(* PLC project Horosheva_14_20160824, CODESYS CODESYS V3.5 SP21 *)
(* stored: creationDateTime 2025-03-30T00:33:44.49212, version 0.0.0.107, modificationDateTime 2025-03-30T00:32:10.5601067 *)

TYPE VLV : STRUCT
  CW : VLV_CW;
  SW : VLV_SW;
  rSetPos : REAL;
  rActPos : REAL;
  wStatus : WORD;
  res7 : INT;
  res8 : INT;
  res9 : INT;
  res10 : INT;
  res11 : INT;
  res12 : INT;
  res13 : INT;
  res14 : INT;
  res15 : INT;
END_STRUCT;
END_TYPE

TYPE MTR : STRUCT
  CW : MTR_CW;
  SW : MTR_SW;
  rMinFreq : REAL;
  rMaxFreq : REAL;
  rManFreq : REAL;
  rAutoFreq : REAL;
  rActFreq : REAL;
  rCurrent : REAL;
  rRunHours : REAL;
  rkWhCount : REAL;
  enStatus : MTR_Stat;
  wFC_StatusWord : WORD;
  dwFC_AlarmWord : DWORD;
  dwFC_WarnWord : DWORD;
  wFC_ErrCode : WORD;
  wIndex : WORD;
  rPower : REAL;
  rHeatsinkTemp : REAL;
  res3 : REAL;
END_STRUCT;
END_TYPE

TYPE SNSR_SW : STRUCT
  Fault : BIT;
  HH_alarm : BIT;
  HL_alarm : BIT;
  LH_alarm : BIT;
  LL_alarm : BIT;
  res5 : BIT;
  res6 : BIT;
  res7 : BIT;
  res8 : BIT;
  res9 : BIT;
  res10 : BIT;
  res11 : BIT;
  res12 : BIT;
  res13 : BIT;
  res14 : BIT;
  res15 : BIT;
END_STRUCT;
END_TYPE

TYPE SNSR_CW : STRUCT
  LimEn : BIT;
  FltrEn : BIT;
  SimEn : BIT;
  ExtFault : BIT;
  res4 : BIT;
  res5 : BIT;
  res6 : BIT;
  res7 : BIT;
  bar_kgf : BIT;
  res9 : BIT;
  res10 : BIT;
  res11 : BIT;
  res12 : BIT;
  res13 : BIT;
  res14 : BIT;
  res15 : BIT;
END_STRUCT;
END_TYPE

TYPE SNSR : STRUCT
  CW : SNSR_CW;
  SW : SNSR_SW;
  k : REAL;
  b : REAL;
  ADC_Range : INT;
  SamplingTime : INT;
  HH : REAL;
  HL : REAL;
  LH : REAL;
  LL : REAL;
  DeadBand : REAL;
  LimDelay : INT;
  res19 : INT;
  res20 : INT;
  res21 : INT;
  PIW : INT;
  IntValue : INT;
  RealValue : REAL;
  SimValue : REAL;
  AccumDir : REAL;
  AccumRev : REAL;
END_STRUCT;
END_TYPE

TYPE VLV_SW : STRUCT
  xRem : BIT;
  xManAuto : BIT;
  xCOM_Open : BIT;
  xCOM_Close : BIT;
  xRUN : BIT;
  xOpened : BIT;
  xClosed : BIT;
  xAlarmAccum : BIT;
  xManOK : BIT;
  xAutoOK : BIT;
  xRunManual : BIT;
  xRunAuto : BIT;
  res12 : BIT;
  res13 : BIT;
  res14 : BIT;
  res15 : BIT;
END_STRUCT;
END_TYPE

(* values of VLV_Stat: STANDBY: Standby; OPENED: Opened; CLOSED: Closed; ALARM_ACCUM: Alarm; BLOCK: Blocked (QM off or smth. else) *)

TYPE VLV_Stat : (STANDBY := 0, OPENED := 1, CLOSED := 2, ALARM_ACCUM := 3, BLOCK := 4);
END_TYPE

TYPE VLV_CW : STRUCT
  xEnable : BIT;
  xAuxON : BIT;
  xExtraAlarm : BIT;
  xACK : BIT;
  xAutoMode : BIT;
  xManMode : BIT;
  xManOpen : BIT;
  xStop : BIT;
  xManClose : BIT;
  xAutoOpen : BIT;
  xAutoClose : BIT;
  xExtraEn : BIT;
  res12 : BIT;
  res13 : BIT;
  res14 : BIT;
  xSimEn : BIT;
END_STRUCT;
END_TYPE

(* values of MTR_Stat: STANDBY: Standby; RUN_MAN: Work in manual mode; STAND_MAN: Stand in manual mode; RUN_AUTO: Work in auto mode; STAND_AUTO: Stand in auto mode; NOT_IN_CYCLE: In auto mode, but not in auto cycle; ALARM_ACCUM: Alarm; BLOCK: Blocked (QM off or smth. else) *)

(* -----Motor status-----// *)
TYPE MTR_Stat : (STANDBY := 0, RUN_MAN := 1, STAND_MAN := 2, RUN_AUTO := 3, STAND_AUTO := 5, NOT_IN_CYCLE := 4, ALARM_ACCUM := 6, BLOCK := 7);
END_TYPE

TYPE MTR_CW : STRUCT
  xEnable : BIT;
  xAuxON : BIT;
  xExtraAlarm : BIT;
  xACK : BIT;
  xAutoMode : BIT;
  xManMode : BIT;
  xManStart : BIT;
  xManStop : BIT;
  xAutoON : BIT;
  xExtraEn : BIT;
  res10 : BIT;
  res11 : BIT;
  res12 : BIT;
  res13 : BIT;
  res14 : BIT;
  xSimEn : BIT;
END_STRUCT;
END_TYPE

TYPE MTR_SW : STRUCT
  xRem : BIT;
  xManAuto : BIT;
  xRUN : BIT;
  xCOM : BIT;
  xAlarmAccum : BIT;
  xReady : BIT;
  res6 : BIT;
  res7 : BIT;
  xManOK : BIT;
  xAutoOK : BIT;
  xRunManual : BIT;
  xRunAuto : BIT;
  res12 : BIT;
  res13 : BIT;
  res14 : BIT;
  res15 : BIT;
END_STRUCT;
END_TYPE

TYPE CCL_WRN : STRUCT
  xVoltageOK : BIT;
  xPLC_ConectOK : BIT;
  xSecurity : BIT;
  xFire : BIT;
  xFireEqipFault : BIT;
  xDrainLL : BIT;
  xDrainHL : BIT;
  xDrainHH : BIT;
  xPMP1_Dry : BIT;
  xPMP2_Dry : BIT;
  xPMP3_Dry : BIT;
  res11 : BIT;
  res12 : BIT;
  res13 : BIT;
  res14 : BIT;
  res15 : BIT;
  res16 : BIT;
  res17 : BIT;
  res18 : BIT;
  res19 : BIT;
  res20 : BIT;
  res21 : BIT;
  res22 : BIT;
  res23 : BIT;
  res24 : BIT;
  res25 : BIT;
  res26 : BIT;
  res27 : BIT;
  res28 : BIT;
  res29 : BIT;
  res30 : BIT;
  res31 : BIT;
END_STRUCT;
END_TYPE

TYPE CCL : STRUCT
  CW : CCL_CW;
  SW : CCL_SW;
  WRN : CCL_WRN;
  uiRotHour : UINT;
  uiRotMin : UINT;
  res6 : WORD;
  res7 : WORD;
  rSP : REAL;
  PmpConnFreq : REAL;
  PmpDisconnFreq : REAL;
  res11 : REAL;
END_STRUCT;
END_TYPE

TYPE CCL_SW : STRUCT
  xALARM : BIT;
  xON : BIT;
  xRunning : BIT;
  res3 : BIT;
  res4 : BIT;
  res5 : BIT;
  res6 : BIT;
  res7 : BIT;
  res8 : BIT;
  res9 : BIT;
  res10 : BIT;
  res11 : BIT;
  res12 : BIT;
  res13 : BIT;
  res14 : BIT;
  res15 : BIT;
END_STRUCT;
END_TYPE

TYPE CCL_CW : STRUCT
  xAuxON : BIT;
  xStart : BIT;
  xStop : BIT;
  xPulseStart : BIT;
  xACK : BIT;
  res5 : BIT;
  res6 : BIT;
  res7 : BIT;
  xAuxStop : BIT;
  xPmpRot : BIT;
  res10 : BIT;
  res11 : BIT;
  res12 : BIT;
  res13 : BIT;
  res14 : BIT;
  res15 : BIT;
END_STRUCT;
END_TYPE

TYPE PID_SW : STRUCT
  Error : BIT;
  LL : BIT;
  LH : BIT;
  res3 : BIT;
  res4 : BIT;
  res5 : BIT;
  res6 : BIT;
  res7 : BIT;
  res8 : BIT;
  res9 : BIT;
  res10 : BIT;
  res11 : BIT;
  res12 : BIT;
  res13 : BIT;
  res14 : BIT;
  res15 : BIT;
END_STRUCT;
END_TYPE

TYPE PID_CW : STRUCT
  En : BIT;
  ManMode : BIT;
  Reset : BIT;
  Hold : BIT;
  res4 : BIT;
  res5 : BIT;
  res6 : BIT;
  res7 : BIT;
  res8 : BIT;
  res9 : BIT;
  res10 : BIT;
  res11 : BIT;
  res12 : BIT;
  res13 : BIT;
  res14 : BIT;
  res15 : BIT;
END_STRUCT;
END_TYPE

TYPE PID_ : STRUCT
  CW : PID_CW;
  SW : PID_SW;
  SetPoint : REAL;
  Kp : REAL;
  Tn : REAL;
  Tv : REAL;
  Td : REAL;
  Offset : REAL;
  ManVal : REAL;
  LL : REAL;
  LH : REAL;
  Y : REAL;
  DIFF : REAL;
  ActValue : REAL;
  DeadBand : REAL;
  MinStop : TIME;
  MinWork : TIME;
END_STRUCT;
END_TYPE

TYPE SP_SW : STRUCT
  xManual : BIT;
  xSched : BIT;
  xRemote : BIT;
  res3 : BIT;
  res4 : BIT;
  res5 : BIT;
  res6 : BIT;
  res7 : BIT;
  res8 : BIT;
  res9 : BIT;
  res10 : BIT;
  res11 : BIT;
  res12 : BIT;
  res13 : BIT;
  res14 : BIT;
  res15 : BIT;
END_STRUCT;
END_TYPE

TYPE SP : STRUCT
  CW : SP_CW;
  SW : SP_SW;
  wSPLocSetNum : WORD;
  wSPLocCurrNum : WORD;
  sSPDate : SP_Date;
  sSPLocSet : SP_Loc;
  arrSPLocCurr : ARRAY[1..4] OF SP_Loc;
  rSPRem : REAL;
  wConnect : WORD;
  wSPRemSet : WORD;
END_STRUCT;
END_TYPE

TYPE SP_Loc : STRUCT
  wHour : WORD;
  wMinute : WORD;
  rSP : REAL;
END_STRUCT;
END_TYPE

TYPE SP_Date : STRUCT
  wSummMonth : WORD;
  wSummDay : WORD;
  wWinMonth : WORD;
  wWinDay : WORD;
END_STRUCT;
END_TYPE

TYPE SP_CW : STRUCT
  xManMode : BIT;
  xAutoLocMode : BIT;
  xAutoRemMode : BIT;
  xConnect : BIT;
  xSPLocSet : BIT;
  xSPRemSet : BIT;
  res6 : BIT;
  res7 : BIT;
  res8 : BIT;
  res9 : BIT;
  res10 : BIT;
  res11 : BIT;
  res12 : BIT;
  res13 : BIT;
  res14 : BIT;
  res15 : BIT;
END_STRUCT;
END_TYPE

VAR_GLOBAL  (* GVL *)
  i_write_set_point_Pump : BOOL;
  ETH_Set_ip : SEC_ETH_UTIL.changeIPAddress;
  wSecond AT %MW41605 : UINT;
  wYear AT %MW41600 : UINT;
  wMonth AT %MW41601 : UINT;
  wDay AT %MW41602 : UINT;
  wHour AT %MW41603 : UINT;
  wMinute AT %MW41604 : UINT;
  x_Set_ip : BOOL;
  x_Save_ip : BOOL;
  xPLC_RUN : BOOL;
  i_ADC_Range : INT := 10000;
  PLC_Cycle : REAL := 0.1;
  i_Set_Point_Pressure AT %MD576 : REAL;
  i_input_ip_address AT %MB500 : ARRAY[1..4] OF BYTE;
  FirstCycle : BOOL;
END_VAR

PROGRAM CycleSect
  VAR
    PLC_RUN : BOOL;
    CycleDelay : TON;
    PulseStart : R_TRIG;
    xVoltageOK : BOOL;
    xExtAlarm : BOOL;
    PLS_RESET : R_TRIG;
  END_VAR

            
PLC_RUN:= (PLC_R.i_wStatus = 16#0002);
PLS_RESET(CLK:= PLC_RUN);

Cycle.CW.xAuxON:= PLC_RUN;
Cycle.SW.xON:= (Cycle.CW.xStart OR Cycle.SW.xON) AND NOT Cycle.CW.xAuxStop;  

CycleDelay(IN:= Cycle.SW.xON,PT:= T#3S);
PulseStart(CLK:= CycleDelay.Q AND (Cycle.CW.xStart OR NOT Cycle.SW.xRunning), Q=> Cycle.CW.xPulseStart);

Cycle.SW.xRunning:= CycleDelay.Q;
				
Cycle.CW.xStart:= FALSE;
IF Cycle.CW.xAuxStop THEN
	Cycle.CW.xStop:= FALSE;
	Cycle.CW.xAuxStop:= FALSE;
END_IF



          
END_PROGRAM

PROGRAM CtrlSect
  VAR
    xPMP2_StartRdy : BOOL;
    xPMP3_StartRdy : BOOL;
    xPMP1_StartRdy : BOOL;
    xPMP1_StopRdy : BOOL;
    xPMP2_StopRdy : BOOL;
    xPMP3_StopRdy : BOOL;
    StartPulse : R_TRIG;
    AuxPmpOnTmr : TON;
    AuxPmpOnPls : R_TRIG;
    xStartAuxPmpReq : BOOL;
    AuxPmpOffTmr : TON;
    AuxPmpOffPls : R_TRIG;
    xStopAuxPmpReq : BOOL;
    MainReg : PID;
    AuxReg : PID;
    MainPID_SetFreq : REAL;
    AuxPID_SetFreq : REAL;
    PMP1_Rising : BOOL;
    PMP2_Rising : BOOL;
    PMP3_Rising : BOOL;
    CyclicSubTimer : TON;
    CyclicSubPls : R_TRIG;
    AuxPmpOnTmrET : TIME;
    AuxPmpOffTmrET : TIME;
    iRunPmpNum : INT;
    MainReg_Ymin : REAL;
    AuxReg_Ymin : REAL;
    RotReq : BOOL;
    ConnPls : R_TRIG;
    DisconnPls : R_TRIG;
  END_VAR

            //=====================================================================================================================//
// Definition of pumps ready to start
//=====================================================================================================================//
xPMP1_StartRdy:= PMP1.SW.xAutoOK AND NOT PMP1.SW.xRUN AND
				((PMP1_WorkTimer[3] <= PMP2_WorkTimer[3]) OR NOT PMP2.SW.xAutoOK OR PMP2.SW.xRUN) AND
				((PMP1_WorkTimer[3] <= PMP3_WorkTimer[3]) OR NOT PMP3.SW.xAutoOK OR PMP3.SW.xRUN);
xPMP2_StartRdy:= PMP2.SW.xAutoOK AND NOT PMP2.SW.xRUN AND
				((PMP2_WorkTimer[3] <= PMP1_WorkTimer[3]) OR NOT PMP1.SW.xAutoOK OR PMP1.SW.xRUN) AND 
				((PMP2_WorkTimer[3] <= PMP3_WorkTimer[3]) OR NOT PMP3.SW.xAutoOK OR PMP3.SW.xRUN);
xPMP3_StartRdy:= PMP3.SW.xAutoOK AND NOT PMP3.SW.xRUN AND 
				((PMP3_WorkTimer[3] <= PMP1_WorkTimer[3]) OR NOT PMP1.SW.xAutoOK OR PMP1.SW.xRUN) AND 
				((PMP3_WorkTimer[3] <= PMP2_WorkTimer[3]) OR NOT PMP2.SW.xAutoOK OR PMP2.SW.xRUN);

//=====================================================================================================================//
// Identifying a pump ready to stop
//=====================================================================================================================//
xPMP1_StopRdy:= PMP1.SW.xAutoOK AND PMP1.SW.xRUN AND 
				((PMP1_WorkTimer[3] >= PMP2_WorkTimer[3]) OR NOT PMP2.SW.xRUN) AND 
				((PMP1_WorkTimer[3] >= PMP3_WorkTimer[3]) OR NOT PMP3.SW.xRUN);
xPMP2_StopRdy:= PMP2.SW.xAutoOK AND PMP2.SW.xRUN AND 
				((PMP2_WorkTimer[3] >= PMP1_WorkTimer[3]) OR NOT PMP1.SW.xRUN) AND 
				((PMP2_WorkTimer[3] >= PMP3_WorkTimer[3]) OR NOT PMP3.SW.xRUN);
xPMP3_StopRdy:= PMP3.SW.xAutoOK AND PMP3.SW.xRUN AND 
				((PMP3_WorkTimer[3] >= PMP1_WorkTimer[3]) OR NOT PMP1.SW.xRUN) AND 
				((PMP3_WorkTimer[3] >= PMP2_WorkTimer[3]) OR NOT PMP2.SW.xRUN);
				
//=====================================================================================================================//
// Determining the number of operating pumps and the minimum output value of the main PID controller
//=====================================================================================================================//
IF (PMP1.SW.xRUN AND PMP1.SW.xAutoOK) AND (PMP2.SW.xRUN AND PMP2.SW.xAutoOK) AND(PMP3.SW.xRUN AND PMP3.SW.xAutoOK) THEN
	MainReg_Ymin:= MAX(MAX(PMP1.rMinFreq, PMP2.rMinFreq), PMP3.rMinFreq);
	iRunPmpNum:= 3;
ELSIF ((PMP1.SW.xRUN AND PMP1.SW.xAutoOK) AND (PMP2.SW.xRUN AND PMP2.SW.xAutoOK)) THEN
	MainReg_Ymin:= MAX(PMP1.rMinFreq, PMP2.rMinFreq);
	iRunPmpNum:= 2;
ELSIF ((PMP1.SW.xRUN AND PMP1.SW.xAutoOK) AND (PMP3.SW.xRUN AND PMP3.SW.xAutoOK)) THEN
	MainReg_Ymin:= MAX(PMP1.rMinFreq, PMP3.rMinFreq);
	iRunPmpNum:= 2; 
ELSIF ((PMP2.SW.xRUN AND PMP2.SW.xAutoOK) AND (PMP3.SW.xRUN AND PMP3.SW.xAutoOK)) THEN
	MainReg_Ymin:= MAX(PMP2.rMinFreq, PMP3.rMinFreq);
	iRunPmpNum:= 2;
ELSIF (PMP1.SW.xRUN AND PMP1.SW.xAutoOK) THEN
	MainReg_Ymin:= PMP1.rMinFreq;
	iRunPmpNum:= 1;
ELSIF (PMP2.SW.xRUN AND PMP2.SW.xAutoOK) THEN
	MainReg_Ymin:= PMP2.rMinFreq;
	iRunPmpNum:= 1;
ELSIF (PMP3.SW.xRUN AND PMP3.SW.xAutoOK) THEN
	MainReg_Ymin:= PMP3.rMinFreq;
	iRunPmpNum:= 1;
ELSE
	MainReg_Ymin:= 25.0;
	iRunPmpNum:= 0;
END_IF
			
//====================================================================================================================//
// Pump start request condition
//====================================================================================================================//
AuxPmpOnTmr(IN:= ((PMP1.rActFreq >= (PMP1.rMaxFreq - 1.0)) OR
				  (PMP2.rActFreq >= (PMP2.rMaxFreq - 1.0)) OR
				  (PMP3.rActFreq >= (PMP3.rMaxFreq - 1.0))) AND (xPMP1_StartRdy OR xPMP2_StartRdy OR xPMP3_StartRdy) AND
				 ((BP01.RealValue + 0.3) <= Cycle.rSP) AND Cycle.SW.xRunning, PT:= T#180S, ET=> AuxPmpOnTmrET);
AuxPmpOnPls(CLK:= AuxPmpOnTmr.Q);
//====================================================================================================================//
// Pump shutdown request condition
//====================================================================================================================//
AuxPmpOffTmr(IN:= (((PMP1.rActFreq < Cycle.PmpDisconnFreq) AND xPMP1_StopRdy) OR
				  ((PMP2.rActFreq < Cycle.PmpDisconnFreq) AND xPMP2_StopRdy) OR
				  ((PMP3.rActFreq < Cycle.PmpDisconnFreq) AND xPMP3_StopRdy)) AND (iRunPmpNum > 1) AND
				  ((BP01.RealValue + 0.2) >= Cycle.rSP) AND Cycle.SW.xRunning, PT:= T#180S, ET=> AuxPmpOffTmrET);
AuxPmpOffPls(CLK:= AuxPmpOffTmr.Q);
//====================================================================================================================//
// Time rotation of pumps
//====================================================================================================================//
IF Cycle.CW.xPmpRot AND (xPMP1_StartRdy OR xPMP2_StartRdy OR xPMP3_StartRdy) AND (PLC_RTC.wHour = Cycle.uiRotHour) AND (PLC_RTC.wMinute = Cycle.uiRotMin) AND (PLC_RTC.wSecond = 1) THEN
	RotReq:= TRUE;
END_IF

IF DisconnPls.Q OR NOT Cycle.CW.xPmpRot OR ((PMP1_Rising AND PMP1.SW.xAlarmAccum) OR (PMP2_Rising AND PMP2.SW.xAlarmAccum) OR (PMP3_Rising AND PMP3.SW.xAlarmAccum) AND NOT (xPMP1_StartRdy OR xPMP2_StartRdy OR xPMP3_StartRdy)) THEN
	RotReq:= FALSE;
END_IF

ConnPls(CLK:= RotReq);
DisconnPls(CLK:= RotReq AND (AuxPID.Y >= MainPID.Y));
//====================================================================================================================//
// Generation of pump start-up and shutdown requests
//====================================================================================================================//
StartPulse(CLK:= Cycle.SW.xRunning);
IF Cycle.SW.xRunning THEN
	IF StartPulse.Q OR AuxPmpOnPls.Q OR (iRunPmpNum = 0) OR ConnPls.Q OR (PMP1_Rising AND PMP1.SW.xAlarmAccum) OR (PMP2_Rising AND PMP2.SW.xAlarmAccum) OR (PMP3_Rising AND PMP3.SW.xAlarmAccum) THEN
		xStartAuxPmpReq:= TRUE;
	END_IF

	IF (AuxPmpOffPls.Q OR DisconnPls.Q) AND (iRunPmpNum > 1) THEN
		xStopAuxPmpReq:= TRUE;
	END_IF

ELSE	
	xStartAuxPmpReq:= FALSE;
	xStopAuxPmpReq:= FALSE;
	PMP1.CW.xAutoON:= FALSE;
	PMP2.CW.xAutoON:= FALSE;
	PMP3.CW.xAutoON:= FALSE;
	PMP1_Rising:= FALSE;
	PMP2_Rising:= FALSE;
	PMP3_Rising:= FALSE;
	RotReq:= FALSE;
END_IF

//====================================================================================================================//
// Formation of an acceleration bit on request to start a pump unit or connect an additional pump
//====================================================================================================================//
IF xStartAuxPmpReq THEN
	IF xPMP1_StartRdy THEN
		PMP1_Rising:= TRUE;
	ELSIF xPMP2_StartRdy THEN
		PMP2_Rising:= TRUE;
	ELSIF xPMP3_StartRdy THEN
		PMP3_Rising:= TRUE;
	END_IF
	xStartAuxPmpReq:= FALSE;
END_IF
//====================================================================================================================//
// Setpoint reduction on acceleration
//====================================================================================================================//
IF PMP1_Rising OR PMP2_Rising OR PMP3_Rising THEN
	MainPID.SetPoint:= Cycle.rSP - 1.0;			
	AuxPID.SetPoint:= Cycle.rSP;				
ELSE
	MainPID.SetPoint:= Cycle.rSP;
	AuxPID.SetPoint:= 0.0;
END_IF
//====================================================================================================================//
// Pump No. 1 run-up
//====================================================================================================================// 	
IF PMP1_Rising THEN														
	PMP1.CW.xAutoON:= TRUE;													
	PMP1.rAutoFreq:= AuxPID_SetFreq;										
	                                                                              
	IF AuxPID.Y >= MainPID.Y OR PMP1.SW.xAlarmAccum THEN					
		PMP1_Rising:= FALSE;												
	END_IF                                                                        
ELSIF NOT (xStopAuxPmpReq AND xPMP1_StopRdy) AND NOT Cycle.CW.xStop THEN	 
	PMP1.rAutoFreq:= MainPID_SetFreq;										
END_IF
//====================================================================================================================//
// Pump No. 2 run-up
//====================================================================================================================//
IF PMP2_Rising THEN
	PMP2.CW.xAutoON:= TRUE;
	PMP2.rAutoFreq:= AuxPID_SetFreq;		
	
	IF AuxPID.Y >= MainPID.Y OR PMP2.SW.xAlarmAccum THEN
		PMP2_Rising:= FALSE;
	END_IF
ELSIF NOT (xStopAuxPmpReq AND xPMP2_StopRdy) AND NOT Cycle.CW.xStop THEN
	PMP2.rAutoFreq:= MainPID_SetFreq;
END_IF
//====================================================================================================================//
// Pump No. 3 run-up
//====================================================================================================================//
IF PMP3_Rising THEN
	PMP3.CW.xAutoON:= TRUE;
	PMP3.rAutoFreq:= AuxPID_SetFreq;		

	IF AuxPID.Y >= MainPID.Y OR PMP3.SW.xAlarmAccum THEN
		PMP3_Rising:= FALSE;
	END_IF
ELSIF NOT (xStopAuxPmpReq AND xPMP3_StopRdy) AND NOT Cycle.CW.xStop THEN
	PMP3.rAutoFreq:= MainPID_SetFreq;
END_IF

//====================================================================================================================//
// Smooth stop of redundant pump
//====================================================================================================================//
CyclicSubTimer(IN:= NOT CyclicSubTimer.Q, PT:= T#5S);
CyclicSubPls(CLK:= CyclicSubTimer.Q);

IF xStopAuxPmpReq  THEN
	IF xPMP1_StopRdy THEN
		IF CyclicSubPls.Q THEN
			PMP1.rAutoFreq:= PMP1.rAutoFreq - 2.0;
		END_IF
		IF PMP1.rActFreq <= PMP1.rMinFreq + 2.0 THEN
			PMP1.CW.xAutoON:= FALSE;
			xStopAuxPmpReq:= FALSE;
		END_IF
	ELSIF xPMP2_StopRdy THEN
		IF CyclicSubPls.Q THEN
			PMP2.rAutoFreq:= PMP2.rAutoFreq - 2.0;
		END_IF
		IF PMP2.rActFreq <= PMP2.rMinFreq + 2.0 THEN
			PMP2.CW.xAutoON:= FALSE;
			xStopAuxPmpReq:= FALSE;
		END_IF
	ELSIF xPMP3_StopRdy THEN
		IF CyclicSubPls.Q THEN
			PMP3.rAutoFreq:= PMP3.rAutoFreq - 2.0;
		END_IF
		IF PMP3.rActFreq <= PMP3.rMinFreq + 2.0 THEN
			PMP3.CW.xAutoON:= FALSE;
			xStopAuxPmpReq:= FALSE;
		END_IF
	END_IF
END_IF

//====================================================================================================================//
// Resetting the start command in automatic cycle if the pump is not in automatic mode
//====================================================================================================================//
IF NOT PMP1.SW.xAutoOK THEN
	PMP1.CW.xAutoON:= FALSE;
END_IF	
IF NOT PMP2.SW.xAutoOK THEN
	PMP2.CW.xAutoON:= FALSE;
END_IF	
IF NOT PMP3.SW.xAutoOK THEN
	PMP3.CW.xAutoON:= FALSE;
END_IF	

//====================================================================================================================//
// Soft stop of pumps to disable automatic cycle
//====================================================================================================================//
IF Cycle.CW.xStop AND Cycle.SW.xRunning THEN
	xStartAuxPmpReq:= FALSE;
	xStopAuxPmpReq:= FALSE;
	IF CyclicSubPls.Q THEN
		PMP1.rAutoFreq:= PMP1.rAutoFreq - 2.0;
		PMP2.rAutoFreq:= PMP2.rAutoFreq - 2.0;
		PMP3.rAutoFreq:= PMP3.rAutoFreq - 2.0;
	END_IF
	
	IF ((PMP1.rActFreq <= PMP1.rMinFreq + 2.0) OR NOT PMP1.SW.xAutoOK) AND 
		((PMP2.rActFreq <= PMP2.rMinFreq + 2.0) OR NOT PMP2.SW.xAutoOK) AND 
		((PMP3.rActFreq <= PMP3.rMinFreq + 2.0) OR NOT PMP3.SW.xAutoOK) THEN
		Cycle.CW.xAuxStop:= TRUE;
	END_IF
END_IF

//====================================================================================================================//
// Determining the minimum output value of the auxiliary PID controller
//====================================================================================================================//
IF PMP1_Rising THEN
	AuxReg_Ymin:= PMP1.rMinFreq;
ELSIF PMP2_Rising THEN
	AuxReg_Ymin:= PMP2.rMinFreq;
ELSIF PMP3_Rising THEN
	AuxReg_Ymin:= PMP3.rMinFreq;
ELSE
	AuxReg_Ymin:= 25.0;
END_IF

//====================================================================================================================//
// Main PID controller
//====================================================================================================================//
MainPID.CW.Reset:= NOT(Cycle.SW.xRunning AND (PMP1.SW.xRunAuto OR PMP2.SW.xRunAuto OR PMP3.SW.xRunAuto));
MainPID.ActValue:= BP01.RealValue;
MainReg(
	ACTUAL:= MainPID.ActValue, 
	SET_POINT:= MainPID.SetPoint, 
	KP:= MainPID.Kp, 
	TN:= MainPID.Tn, 
	TV:= MainPID.Tv, 
	Y_MANUAL:= MainPID.ManVal, 
	Y_OFFSET:= MainPID.Offset, 
	Y_MIN:= MainReg_Ymin * 10.0,
	Y_MAX:= 500.0, 
	MANUAL:= MainPID.CW.ManMode, 
	RESET:= MainPID.CW.Reset, 
	Y=> MainPID.Y, 
	LIMITS_ACTIVE=> , 
	OVERFLOW=> );
MainPID_SetFreq:= MainPID.Y / 10.0; 

//====================================================================================================================//
// Auxiliary PID controller used to accelerate the auxiliary pump
//====================================================================================================================//	
AuxPID.CW.Reset:= NOT(Cycle.SW.xRunning AND (PMP1_Rising OR PMP2_Rising OR PMP3_Rising));	
AuxPID.ActValue:= BP01.RealValue;
AuxReg(
	ACTUAL:= AuxPID.ActValue, 
	SET_POINT:= AuxPID.SetPoint, 
	KP:= AuxPID.Kp, 
	TN:= AuxPID.Tn, 
	TV:= AuxPID.Tv, 
	Y_MANUAL:= AuxPID.ManVal, 
	Y_OFFSET:= AuxPID.Offset, 
	Y_MIN:= AuxReg_Ymin * 10.0,
	Y_MAX:= 500.0, 
	MANUAL:= AuxPID.CW.ManMode, 
	RESET:= AuxPID.CW.Reset, 
	Y=> AuxPID.Y, 
	LIMITS_ACTIVE=> , 
	OVERFLOW=> );
AuxPID_SetFreq:= AuxPID.Y / 10.0;
	
	
	
	
	
	
	
	
          
END_PROGRAM

FUNCTION_BLOCK MotorFB
  VAR_INPUT
    SetOvertime : TIME;
    Cycle : CCL;
  END_VAR
  VAR_OUTPUT
    rFreqValue : REAL;
    WorkTime : ARRAY[1..4] OF UDINT;
  END_VAR
  VAR_IN_OUT
    Mot_strct : MTR;
  END_VAR
  VAR
    TON_Overtime : TON;
    xAlarmFeedback : BOOL;
    xEnableMotorAuto : BOOL;
    xCOM : BOOL;
    WTC : WTCount;
    xAlarmBlock : BOOL;
  END_VAR

            	(*Alarm Feedback processing*)
TON_Overtime(IN:=Mot_strct.CW.xEnable AND ((Mot_strct.SW.xCOM AND NOT Mot_strct.SW.xRUN) OR (NOT Mot_strct.SW.xCOM AND Mot_strct.SW.xRUN)),PT:=SetOvertime);

IF TON_Overtime.Q THEN
	xAlarmFeedback:=TRUE;
END_IF; 

IF NOT Mot_strct.CW.xExtraEn AND xCOM THEN
	xAlarmBlock:= TRUE;
END_IF

Mot_strct.SW.xAlarmAccum:= xAlarmFeedback OR Mot_strct.CW.xExtraAlarm OR xAlarmBlock;

IF Mot_strct.CW.xACK THEN
	xAlarmFeedback:= FALSE;
	xAlarmBlock:= FALSE;
END_IF
	
	(*Auto/Manual mode selection*)
IF Mot_strct.CW.xAutoMode THEN
	xEnableMotorAuto:= TRUE;
ELSIF Mot_strct.CW.xManMode THEN
	xEnableMotorAuto:= FALSE;
END_IF;
Mot_strct.SW.xManAuto:= xEnableMotorAuto; 

Mot_strct.SW.xManOK:= NOT Mot_strct.SW.xAlarmAccum AND Mot_strct.CW.xAuxON AND Mot_strct.CW.xEnable AND NOT xEnableMotorAuto;
Mot_strct.SW.xAutoOK:= NOT Mot_strct.SW.xAlarmAccum AND Mot_strct.CW.xAuxON AND Mot_strct.CW.xEnable AND xEnableMotorAuto;

	(*Motor ready to start*)
Mot_strct.SW.xReady:= (Mot_strct.SW.xManOK OR Mot_strct.SW.xAutoOK) AND NOT Mot_strct.SW.xAlarmAccum;

	(*Manual mode activation*)
IF Mot_strct.CW.xManStart THEN
	Mot_strct.SW.xRunManual:=TRUE;
END_IF;
IF Mot_strct.CW.xManStop OR NOT Mot_strct.SW.xManOK THEN
	Mot_strct.SW.xRunManual:=FALSE;
END_IF;

	(*Auto mode activation*)
Mot_strct.SW.xRunAuto:= Mot_strct.SW.xAutoOK AND Cycle.SW.xRunning;

	(*Set command for start*)
xCOM:=((Mot_strct.SW.xRunManual AND Mot_strct.SW.xManOK) OR (Mot_strct.SW.xRunAuto AND Mot_strct.SW.xAutoOK AND Mot_strct.CW.xAutoON));
Mot_strct.SW.xCOM:= xCOM AND NOT Mot_strct.CW.xSimEn;

	(*Work time counter*)
WTC(StartCount:= Mot_strct.SW.xRUN, udiSeconds=> WorkTime[4], udiMinutes=> WorkTime[3], udiHours=> WorkTime[2], udiDays=> WorkTime[1]);

	(*Frequency limitation*)
Mot_strct.rMaxFreq:= LIMIT(0.0, Mot_strct.rMaxFreq, 50.0);
Mot_strct.rMinFreq:= LIMIT(0.0, Mot_strct.rMinFreq, Mot_strct.rMaxFreq);	
Mot_strct.rManFreq:= LIMIT(Mot_strct.rMinFreq, Mot_strct.rManFreq, Mot_strct.rMaxFreq);
Mot_strct.rAutoFreq:= LIMIT(Mot_strct.rMinFreq, Mot_strct.rAutoFreq, Mot_strct.rMaxFreq);

IF Mot_strct.SW.xRunAuto THEN
	rFreqValue:= Mot_strct.rAutoFreq;
ELSIF Mot_strct.SW.xRunManual THEN
	rFreqValue:= Mot_strct.rManFreq;
ELSE
	rFreqValue:= 0.0;
END_IF;

	(*Status processing*)
IF Mot_strct.SW.xAlarmAccum THEN											//Alarm
	Mot_strct.enStatus:= MTR_Stat.ALARM_ACCUM;
ELSIF Mot_strct.SW.xCOM AND Mot_strct.SW.xRunManual THEN					//Work in manual mode
	Mot_strct.enStatus:= MTR_Stat.RUN_MAN;
ELSIF Mot_strct.SW.xManOK THEN												//Stand in manual mode
	Mot_strct.enStatus:= MTR_Stat.STAND_MAN;	
ELSIF Mot_strct.SW.xCOM AND Mot_strct.SW.xRunAuto THEN						//Work in auto mode
	Mot_strct.enStatus:= MTR_Stat.RUN_AUTO;
ELSIF Mot_strct.SW.xRunAuto THEN											//Stand in auto mode
	Mot_strct.enStatus:= MTR_Stat.STAND_AUTO;
ELSIF Mot_strct.SW.xAutoOK THEN												//In auto mode, but not in auto cycle
	Mot_strct.enStatus:= MTR_Stat.NOT_IN_CYCLE;			
ELSIF NOT Mot_strct.CW.xExtraEn THEN										//Block
	Mot_strct.enStatus:= MTR_Stat.BLOCK ;					
ELSE																		//Standby
	Mot_strct.enStatus:= MTR_Stat.STANDBY;								
END_IF;

Mot_strct.CW.xAutoMode:= FALSE;
Mot_strct.CW.xManMode:= FALSE;
Mot_strct.CW.xManStart:= FALSE;
Mot_strct.CW.xManStop:= FALSE;
Mot_strct.CW.xACK:= FALSE;
          
END_FUNCTION_BLOCK

FUNCTION_BLOCK WTCount
  VAR_INPUT
    StartCount : BOOL;
  END_VAR
  VAR_OUTPUT
    udiSeconds : UDINT;
    udiMinutes : UDINT;
    udiHours : UDINT;
    udiDays : UDINT;
  END_VAR
  VAR RETAIN PERSISTENT
    udiCount : UDINT;
  END_VAR
  VAR
    PLS : F_TRIG;
  END_VAR

            
	//Work time counter
PLS(CLK:= PLC_R.i_x1sClk);
IF StartCount AND PLS.Q THEN
	udiCount:= udiCount + 1;
END_IF

udiSeconds:= udiCount;
udiMinutes:= udiSeconds / 60;
udiHours:= udiSeconds / 3600;
udiDays:= udiSeconds / 86400;

          
END_FUNCTION_BLOCK

PROGRAM AlarmSect
  VAR
    PLS_Restart : R_TRIG;
    TON_Restart : TON;
  END_VAR

            
Cycle.SW.xALARM:= PMP1.SW.xAlarmAccum OR 
				PMP2.SW.xAlarmAccum OR 
				PMP3.SW.xAlarmAccum OR
				NOT Cycle.WRN.xVoltageOK;

(*TON_Restart(IN:= Cycle.SW.xRunning AND Cycle.WRN.xVoltageOK, PT:= T#3S);				
PLS_Restart(CLK:= TON_Restart.Q);*)	
				
IF Cycle.CW.xACK OR ixACK OR PLS_Restart.Q THEN
	PMP1.CW.xACK:= TRUE;
	PMP2.CW.xACK:= TRUE;
	PMP3.CW.xACK:= TRUE;
	Cycle.WRN.xPMP1_Dry:= FALSE;
	Cycle.WRN.xPMP2_Dry:= FALSE;
	Cycle.WRN.xPMP3_Dry:= FALSE;
	Cycle.CW.xACK:= FALSE;
END_IF
          
END_PROGRAM

PROGRAM TimeSync
  VAR
    NTP_Data : ReadNTPData;
    xAuto : BOOL := TRUE;
    xSync : BOOL := TRUE;
    Err : UDINT;
    xManPing : BOOL;
  END_VAR

            
NTP_Data(
	xAuto:= xAuto, 
	xSync:= xSync, 
	tSync:= T#1H, 
	IP_addr:= '172.16.34.34', 
	iBias:= 4, 
	xPing:= xManPing, 
	ServerDate=> ServerTime, 
	PLC_time=> PLC_RTC, 
	eError=> Err, 
	xNTPSynchronously=> );

          
END_PROGRAM

PROGRAM DI_DO
  VAR
    A00_IW : WORD_AS_BIT;
    A01 : WORD_AS_BIT;
    A00_QW : BIT_AS_WORD;
    A02 : BIT_AS_WORD;
    VoltageOK_1 : BOOL;
    VoltageOK_2 : BOOL;
  END_VAR

            A00_IW(
	W:= iwDI_IW0, 
	B00=> VoltageOK_1, 
	B01=> , 
	B02=> , 
	B03=> , 
	B04=> ,
	B05=> ,
	B06=> , 
	B07=> , 
	B08=> , 
	B09=> , 
	B10=> , 
	B11=> , 
	B12=> , 
	B13=> , 
	B14=> , 
	B15=> );
	
A00_QW(
	B00:= ,
	B01:= , 
	B02:= , 
	B03:= , 
	B04:= Cycle.SW.xALARM, 
	B05:= , 
	B06:= , 
	B07:= , 
	B08:= , 
	B09:= , 
	B10:= , 
	B11:= , 
	B12:= , 
	B13:= , 
	B14:= , 
	B15:= , 
	W=> qwDQ_QW0);


A01(
	W:= iwA01_IW0, 
	B00=> VoltageOK_2, 
	B01=> ixACK, 
	B02=> PMP1.SW.xRem, 
	B03=> PMP1.SW.xRUN, 
	B04=> PMP2.SW.xRem,
	B05=> PMP2.SW.xRUN,
	B06=> PMP3.SW.xRem, 
	B07=> PMP3.SW.xRUN, 
	B08=> Cycle.WRN.xDrainLL, 
	B09=> Cycle.WRN.xDrainHL, 
	B10=> Cycle.WRN.xDrainHH, 
	B11=> , 
	B12=> , 
	B13=> , 
	B14=> Cycle.WRN.xFire, 
	B15=> Cycle.WRN.xFireEqipFault);	
	
A02(
	B00:= Cycle.SW.xALARM, 					//Alarm Lamp
	B01:= Cycle.WRN.xPLC_ConectOK, 
	B02:= PMP1.SW.xCOM, 
	B03:= PMP2.SW.xCOM, 
	B04:= PMP3.SW.xCOM, 
	B05:= , 
	B06:= , 
	B07:= , 
	B08:= , 
	B09:= , 
	B10:= , 
	B11:= , 
	B12:= , 
	B13:= , 
	B14:= , 
	B15:= , 
	W=> qwA02_QB0);
	
Cycle.WRN.xVoltageOK:= VoltageOK_1 AND VoltageOK_2;	
Cycle.WRN.xPLC_ConectOK:= plc_r.i_lwSystemFault_1.1;

          
END_PROGRAM

PROGRAM MotorSect
  VAR
    PMP1_FB : MotorFB;
    PMP2_FB : MotorFB;
    PMP3_FB : MotorFB;
    PMP_DRAIN_FB : MotorFB;
    VFD1_REF_SCALLING : LIN_TRAFO;
    VFD2_REF_SCALLING : LIN_TRAFO;
    VFD3_REF_SCALLING : LIN_TRAFO;
    rVFD1_SetFreq : REAL;
    rVFD2_SetFreq : REAL;
    rVFD3_SetFreq : REAL;
  END_VAR

            
PMP1.CW.xAuxON:= Cycle.CW.xAuxON;
PMP1.CW.xEnable:= PMP1.SW.xRem;
PMP1.CW.xExtraAlarm:= Cycle.WRN.xPMP1_Dry OR (PMP1.dwFC_AlarmWord <> 0);
PMP1.CW.xExtraEn:= TRUE;
PMP1_FB(
	SetOvertime:= T#10S, 
	Cycle:= Cycle, 
	rFreqValue=> , 
	WorkTime=> PMP1_WorkTimer, 
	Mot_strct:= PMP1);
PMP1.rActFreq:= WORD_TO_REAL(wFreq_VFD_1) / 10.0;
PMP1.rCurrent:= WORD_TO_REAL(wI_VFD_1) / 100.0;
PMP1.rPower:= WORD_TO_REAL(wPower_VFD_1) / 1000.0;
PMP1.rRunHours:= DWORD_TO_REAL(MEM.PackWordsToDword(wHighWord:= CountWork_VFD_1_1, wLowWord:= CountWork_VFD_1_2));
PMP1.rkWhCount:= DWORD_TO_REAL(MEM.PackWordsToDword(wHighWord:= wEnergyCount_VFD_1_1, wLowWord:= wEnergyCount_VFD_1_2));
PMP1.wFC_StatusWord:= wStatus_VFD_1;
PMP1.dwFC_AlarmWord:= MEM.PackWordsToDword(wHighWord:= wFault_VFD_1_1, wLowWord:= wFault_VFD_1_2);
PMP1.rHeatsinkTemp:= WORD_TO_REAL(wT_freq_1);

	
IF PMP1.SW.xManAuto THEN
	rVFD1_SetFreq:= PMP1.rAutoFreq;
ELSE
	rVFD1_SetFreq:= PMP1.rManFreq;
END_IF;	

VFD1_REF_SCALLING(IN:= rVFD1_SetFreq, IN_MIN:= 0.0, IN_MAX:= 50.0, OUT_MIN:= 16#0, OUT_MAX:= 16#4000);	
iFreq_Set_1:= REAL_TO_WORD(VFD1_REF_SCALLING.OUT);

IF BP12.SW.LL_alarm AND PMP1.SW.xRUN THEN
	Cycle.WRN.xPMP1_Dry:= TRUE;
END_IF;

	
	

PMP2.CW.xAuxON:= Cycle.CW.xAuxON;	
PMP2.CW.xEnable:= PMP2.SW.xRem;
PMP2.CW.xExtraAlarm:= Cycle.WRN.xPMP2_Dry OR (PMP2.dwFC_AlarmWord <> 0);
PMP2.CW.xExtraEn:= TRUE;
PMP2_FB(
	SetOvertime:= T#10S, 
	Cycle:= Cycle, 
	rFreqValue=> , 
	WorkTime=> PMP2_WorkTimer, 
	Mot_strct:= PMP2);
PMP2.rActFreq:= WORD_TO_REAL(wFreq_VFD_2) / 10.0;
PMP2.rCurrent:= WORD_TO_REAL(wI_VFD_2) / 100.0;
PMP2.rPower:= WORD_TO_REAL(wPower_VFD_2) / 1000.0;
PMP2.rRunHours:= DWORD_TO_REAL(MEM.PackWordsToDword(wHighWord:= CountWork_VFD_2_1, wLowWord:= CountWork_VFD_2_2));
PMP2.rkWhCount:= DWORD_TO_REAL(MEM.PackWordsToDword(wHighWord:= wEnergyCount_VFD_2_1, wLowWord:= wEnergyCount_VFD_2_2));
PMP2.wFC_StatusWord:= wStatus_VFD_2;
PMP2.dwFC_AlarmWord:= MEM.PackWordsToDword(wHighWord:= wFault_VFD_2_1, wLowWord:= wFault_VFD_2_2);
PMP2.rHeatsinkTemp:= WORD_TO_REAL(wT_freq_2);

IF PMP2.SW.xManAuto THEN
	rVFD2_SetFreq:= PMP2.rAutoFreq;
ELSE
	rVFD2_SetFreq:= PMP2.rManFreq;
END_IF;	
VFD2_REF_SCALLING(IN:= rVFD2_SetFreq, IN_MIN:= 0.0, IN_MAX:= 50.0, OUT_MIN:= 16#0, OUT_MAX:= 16#4000);	
iFreq_Set_2:= REAL_TO_WORD(VFD2_REF_SCALLING.OUT);	
	
IF BP22.SW.LL_alarm AND PMP2.SW.xRUN THEN
	Cycle.WRN.xPMP2_Dry:= TRUE;
END_IF;




PMP3.CW.xAuxON:= Cycle.CW.xAuxON;
PMP3.CW.xEnable:= PMP3.SW.xRem;
PMP3.CW.xExtraAlarm:= Cycle.WRN.xPMP3_Dry OR (PMP3.dwFC_AlarmWord <> 0);	
PMP3.CW.xExtraEn:= TRUE;	
PMP3_FB(
	SetOvertime:= T#10S, 
	Cycle:= Cycle, 
	rFreqValue=> , 
	WorkTime=> PMP3_WorkTimer, 
	Mot_strct:= PMP3);
PMP3.rActFreq:= WORD_TO_REAL(wFreq_VFD_3) / 10.0;
PMP3.rCurrent:= WORD_TO_REAL(wI_VFD_3) / 100.0;
PMP3.rPower:= WORD_TO_REAL(wPower_VFD_3) / 1000.0;
PMP3.rRunHours:= DWORD_TO_REAL(MEM.PackWordsToDword(wHighWord:= CountWork_VFD_3_1, wLowWord:= CountWork_VFD_3_2));
PMP3.rkWhCount:= DWORD_TO_REAL(MEM.PackWordsToDword(wHighWord:= wEnergyCount_VFD_3_1, wLowWord:= wEnergyCount_VFD_3_2));
PMP3.wFC_StatusWord:= wStatus_VFD_3;
PMP3.dwFC_AlarmWord:= MEM.PackWordsToDword(wHighWord:= wFault_VFD_3_1, wLowWord:= wFault_VFD_3_2);
PMP3.rHeatsinkTemp:= WORD_TO_REAL(wT_freq_3);

	
IF PMP3.SW.xManAuto THEN
	rVFD3_SetFreq:= PMP3.rAutoFreq;
ELSE
	rVFD3_SetFreq:= PMP3.rManFreq;
END_IF;	
VFD3_REF_SCALLING(IN:= rVFD3_SetFreq, IN_MIN:= 0.0, IN_MAX:= 50.0, OUT_MIN:= 16#0, OUT_MAX:= 16#4000);	
iFreq_Set_3:= REAL_TO_WORD(VFD3_REF_SCALLING.OUT);

IF BP32.SW.LL_alarm AND PMP3.SW.xRUN THEN
	Cycle.WRN.xPMP3_Dry:= TRUE;
END_IF;



(*
PMP_DRAIN.CW.xAuxON:= Cycle.CW.xAuxON;
PMP_DRAIN.CW.xEnable:= PMP_DRAIN.SW.xRem;
PMP_DRAIN.CW.xExtraAlarm:= FALSE;
PMP_DRAIN_FB(
	SetOvertime:= T#5S, 
	Cycle:= Cycle, 
	rFreqValue=> , 
	WorkTime=> PMP_DRAIN_WorkTimer, 
	Mot_strct:= PMP_DRAIN);

*)

          
END_PROGRAM

PROGRAM SensorSect
  VAR
    BP00_FB : SensorFB;
    BP01_FB : SensorFB;
    BP11_FB : SensorFB;
    BP12_FB : SensorFB;
    BP21_FB : SensorFB;
    BP22_FB : SensorFB;
    BP31_FB : SensorFB;
    BP32_FB : SensorFB;
    BT00_FB : SensorFB;
    BL00_FB : SensorFB;
  END_VAR

            
//Output collector pressure
BP00.PIW:= iiA1_1_IW2;
BP00.CW.ExtFault:= (ibA1_1_IBStatusIW2 <> 0);
BP00.k:= 16.0;
BP00.ADC_Range:= 10000;
BP00.CW.bar_kgf:= TRUE;
BP00_FB(Snsr_strct:= BP00);

//Input collector pressure
BP01.PIW:= iiA1_1_IW0;
BP01.CW.ExtFault:= (ibA1_1_IBStatusIW0 <> 0);
BP01.k:= 16.0;
BP01.ADC_Range:= 10000;
BP01.CW.bar_kgf:= TRUE;
BP01_FB(Snsr_strct:= BP01);


//Pump 1 inlet pressure
BP11.PIW:= iiA03_IW0;
BP11.CW.ExtFault:= (ibA03_IBStatusIW0 <> 0);
BP11.k:= 6.0;
BP11.b:= -1.0;
BP11.ADC_Range:= 10000;
BP11.CW.bar_kgf:= TRUE;
BP11.CW.LimEn:= FALSE;
BP11.LL:= 1.0;
BP11.DeadBand:= 0.5;
BP11.LimDelay:= 5;
BP11_FB(Snsr_strct:= BP11);

//Pump 1 outlet pressure
BP12.PIW:= iiA03_IW1;
BP12.CW.ExtFault:= (ibA03_IBStatusIW1 <> 0);
BP12.k:= 10.0;
BP12.ADC_Range:= 10000;
BP12.CW.bar_kgf:= TRUE;
BP12.CW.LimEn:= PMP1.SW.xRUN;
BP12.LL:= BP11.RealValue + 1.0;
BP12.DeadBand:= 0.0;
BP12.LimDelay:= 60;
BP12_FB(Snsr_strct:= BP12);

//Pump 2 inlet pressure
BP21.PIW:= iiA03_IW2;
BP21.CW.ExtFault:= (ibA03_IBStatusIW2 <> 0);
BP21.k:= 6.0;
BP21.b:= -1.0;
BP21.ADC_Range:= 10000;
BP21.CW.bar_kgf:= TRUE;
BP21.CW.LimEn:= FALSE;
BP21.LL:= 1.0;
BP21.DeadBand:= 0.5;
BP21.LimDelay:= 5;
BP21_FB(Snsr_strct:= BP21);

//Pump 2 outlet pressure
BP22.PIW:= iiA03_IW3;
BP22.CW.ExtFault:= (ibA03_IBStatusIW3 <> 0);
BP22.k:= 10.0;
BP22.ADC_Range:= 10000;
BP22.CW.bar_kgf:= TRUE;
BP22.CW.LimEn:= PMP2.SW.xRUN;
BP22.LL:= BP21.RealValue + 1.0;
BP22.DeadBand:= 0.0; 
BP22.LimDelay:= 60;
BP22_FB(Snsr_strct:= BP22);

//Pump 3 inlet pressure
BP31.PIW:= iiA03_IW4;
BP31.CW.ExtFault:= (ibA03_IBStatusIW4 <> 0);
BP31.k:= 6.0;
BP31.b:= -1.0;
BP31.ADC_Range:= 10000;
BP31.CW.bar_kgf:= TRUE;
BP31.CW.LimEn:= FALSE;
BP31.LL:= 1.0;
BP31.DeadBand:= 0.5;
BP31.LimDelay:= 10;
BP31_FB(Snsr_strct:= BP31);

//Pump 3 outlet pressure
BP32.PIW:= iiA03_IW5;
BP32.CW.ExtFault:= (ibA03_IBStatusIW5 <> 0);
BP32.k:= 10.0;
BP32.ADC_Range:= 10000;
BP32.CW.bar_kgf:= TRUE;
BP32.CW.LimEn:= PMP3.SW.xRUN;
BP32.LL:= BP31.RealValue + 1.0;
BP32.DeadBand:= 0.0;
BP32.LimDelay:= 60;
BP32_FB(Snsr_strct:= BP32);


//Tank level
BL00.PIW:= iiA1_1_IW1;
BL00.CW.ExtFault:= (ibA1_1_IBStatusIW1 <> 0);
BL00.k:= 5.0;
BL00.ADC_Range:= 10000;
BL00.CW.bar_kgf:= FALSE;
BL00_FB(Snsr_strct:= BL00);

//Internal temperature
BT00.PIW:= iiA1_1_IW3;
BT00.CW.ExtFault:= (ibA1_1_IBStatusIW3 <> 0);
BT00.k:= 1000.0;
BT00.ADC_Range:= 10000;
BT00.CW.bar_kgf:= FALSE;
BT00_FB(Snsr_strct:= BT00);



          
END_PROGRAM

FUNCTION_BLOCK SensorFB
  VAR
    bar_kgf : REAL;
    RealValue : REAL;
    FltrValue : REAL;
    CycTmr : TON;
    SumValue : REAL;
    Buff : ARRAY[0..9] OF REAL;
    i : INT;
    y : INT;
    INIT : BOOL;
    tonHHTopDelay : TON;
    tonHHBotDelay : TON;
    tonHLTopDelay : TON;
    tonHLBotDelay : TON;
    tonLHTopDelay : TON;
    tonLHBotDelay : TON;
    tonLLTopDelay : TON;
    tonLLBotDelay : TON;
  END_VAR
  VAR_IN_OUT
    Snsr_strct : SNSR;
  END_VAR

            // Fault operation
IF Snsr_strct.PIW < 0 OR Snsr_strct.PIW > Snsr_strct.ADC_Range OR Snsr_strct.CW.ExtFault THEN		(*Snsr_strct Failed*)
	Snsr_strct.SW.Fault:= TRUE;
	RealValue:= 0.0;
ELSE                                                                    			(*Snsr_strct OK*)
	IF Snsr_strct.ADC_Range <= 0 THEN
		Snsr_strct.ADC_Range:= 1;
	END_IF
	Snsr_strct.SW.Fault:= FALSE;
	RealValue:= Snsr_strct.k * bar_kgf * INT_TO_REAL(Snsr_strct.PIW) / INT_TO_REAL(Snsr_strct.ADC_Range) + Snsr_strct.b;	
END_IF

// Converting from bar to kgf/sm2
IF Snsr_strct.CW.bar_kgf THEN
	bar_kgf:= 1.0197;
ELSE
	bar_kgf:= 1.0;
END_IF		


// SMA filter operation
CycTmr(IN:= NOT CycTmr.Q AND INIT, PT:= INT_TO_TIME(Snsr_strct.SamplingTime / 1000));	(*Sample puls generator*)
IF Snsr_strct.CW.FltrEn THEN
	IF NOT INIT THEN																	(*Initialization*)
		FOR y:= 0 TO 9 DO
			Buff[y]:= RealValue;
			SumValue:= SumValue + Buff[y];
		END_FOR
		INIT:= TRUE;
	END_IF
	
	IF CycTmr.Q THEN																	(*Buffer shifting and changing last element*)
		FOR y:= 0 TO 8 DO
			Buff[y]:= Buff[y + 1];
		END_FOR
		Buff[9]:= RealValue;
		SumValue:= SumValue + RealValue - Buff[0];											
	END_IF
	FltrValue:= SumValue / 10;
ELSE
	INIT:= FALSE;
	SumValue:= 0.0;
	FltrValue:= 0.0;
END_IF	

// Snsr_strct output values states
IF Snsr_strct.CW.SimEn THEN															(*Simulated output value*)						
	Snsr_strct.RealValue:= Snsr_strct.SimValue;
	Snsr_strct.IntValue:= REAL_TO_INT(Snsr_strct.SimValue * 100.0);
ELSIF Snsr_strct.CW.FltrEn THEN														(*Filtered output value*)
	Snsr_strct.RealValue:= FltrValue;
	Snsr_strct.IntValue:= REAL_TO_INT(FltrValue * 100.0);
ELSE																				(*Real output value*)
	Snsr_strct.RealValue:= RealValue;
	Snsr_strct.IntValue:= REAL_TO_INT(RealValue * 100.0);
END_IF

// Limits operation
tonHHTopDelay(IN:= (Snsr_strct.RealValue >= Snsr_strct.HH + Snsr_strct.DeadBand / 2.0) AND Snsr_strct.CW.LimEn, PT:= INT_TO_TIME(Snsr_strct.LimDelay * 1000));
tonHHBotDelay(IN:= (Snsr_strct.RealValue <= Snsr_strct.HH - Snsr_strct.DeadBand / 2.0) AND Snsr_strct.CW.LimEn, PT:= INT_TO_TIME(Snsr_strct.LimDelay * 1000));	
tonHLTopDelay(IN:= (Snsr_strct.RealValue >= Snsr_strct.HL + Snsr_strct.DeadBand / 2.0) AND Snsr_strct.CW.LimEn, PT:= INT_TO_TIME(Snsr_strct.LimDelay * 1000));
tonHLBotDelay(IN:= (Snsr_strct.RealValue <= Snsr_strct.HL - Snsr_strct.DeadBand / 2.0) AND Snsr_strct.CW.LimEn, PT:= INT_TO_TIME(Snsr_strct.LimDelay * 1000));

tonLHTopDelay(IN:= (Snsr_strct.RealValue <= Snsr_strct.LH - Snsr_strct.DeadBand / 2.0) AND Snsr_strct.CW.LimEn, PT:= INT_TO_TIME(Snsr_strct.LimDelay * 1000));
tonLHBotDelay(IN:= (Snsr_strct.RealValue >= Snsr_strct.LH + Snsr_strct.DeadBand / 2.0) AND Snsr_strct.CW.LimEn, PT:= INT_TO_TIME(Snsr_strct.LimDelay * 1000));
tonLLTopDelay(IN:= (Snsr_strct.RealValue <= Snsr_strct.LL - Snsr_strct.DeadBand / 2.0) AND Snsr_strct.CW.LimEn, PT:= INT_TO_TIME(Snsr_strct.LimDelay * 1000));
tonLLBotDelay(IN:= (Snsr_strct.RealValue >= Snsr_strct.LL + Snsr_strct.DeadBand / 2.0) AND Snsr_strct.CW.LimEn, PT:= INT_TO_TIME(Snsr_strct.LimDelay * 1000));

IF tonHHTopDelay.Q THEN
	Snsr_strct.SW.HH_alarm:= TRUE;
END_IF	
IF tonHHBotDelay.Q THEN
	Snsr_strct.SW.HH_alarm:= FALSE;
END_IF
IF tonHLTopDelay.Q THEN
	Snsr_strct.SW.HL_alarm:= TRUE;
END_IF
IF tonHLBotDelay.Q THEN
	Snsr_strct.SW.HL_alarm:= FALSE;
END_IF
IF tonLHTopDelay.Q THEN
	Snsr_strct.SW.LH_alarm:= TRUE;
END_IF
IF tonLHBotDelay.Q THEN
	Snsr_strct.SW.LH_alarm:= FALSE;
END_IF
IF tonLLTopDelay.Q THEN
	Snsr_strct.SW.LL_alarm:= TRUE;
END_IF
IF tonLLBotDelay.Q THEN
	Snsr_strct.SW.LL_alarm:= FALSE;
END_IF
	
IF NOT Snsr_strct.CW.LimEn THEN
	Snsr_strct.SW.HH_alarm:= FALSE;
	Snsr_strct.SW.HL_alarm:= FALSE;
	Snsr_strct.SW.LH_alarm:= FALSE;
	Snsr_strct.SW.LL_alarm:= FALSE;	
END_IF

          
END_FUNCTION_BLOCK

FUNCTION_BLOCK ValveFB
  VAR_INPUT
    SetOvertime : TIME;
    Cycle : CCL;
  END_VAR
  VAR_OUTPUT
    COM_Open : BOOL;
    COM_Close : BOOL;
  END_VAR
  VAR
    FeedBackAlrmTmr : TON;
    AlrmNotMove : BOOL;
    AlrmSQ : BOOL;
    AlrmNotMoveTmr : TON;
    AlrmFeedBack : BOOL;
    EnableVlvAuto : BOOL;
    AlarmBlock : BOOL;
  END_VAR
  VAR_IN_OUT
    Vlv_strct : VLV;
  END_VAR

            	//Alarm processing
FeedBackAlrmTmr(IN:= Vlv_strct.CW.xEnable AND (COM_Close OR COM_Open) AND NOT Vlv_strct.SW.xRUN, PT:= T#3S);
AlrmNotMoveTmr(IN:= Vlv_strct.CW.xEnable AND ((COM_Close AND NOT Vlv_strct.SW.xClosed) OR (COM_Open AND NOT Vlv_strct.SW.xOpened), PT:= SetOvertime);

IF FeedBackAlrmTmr.Q THEN 
	AlrmFeedBack:= TRUE;
END_IF

IF AlrmNotMoveTmr.Q THEN 
	AlrmNotMove:= TRUE;
END_IF

IF Vlv_strct.SW.xOpened AND Vlv_strct.SW.xClosed THEN
	AlrmSQ:= TRUE;
END_IF

IF NOT Vlv_strct.CW.xExtraEn AND (COM_Open OR COM_Close) THEN
	AlarmBlock:= TRUE;
END_IF

Vlv_strct.SW.xAlarmAccum:= AlrmFeedBack OR AlrmNotMove OR AlrmSQ OR AlarmBlock OR Vlv_strct.CW.xExtraAlarm; 

IF Vlv_strct.CW.xACK THEN
	AlrmSQ:= FALSE;
	AlrmNotMove:= FALSE;
	AlrmFeedBack:= FALSE;
	AlarmBlock:= FALSE;
END_IF

	//Auto/Manual mode selection
IF Vlv_strct.CW.xAutoMode THEN
	EnableVlvAuto:= TRUE;
END_IF
IF Vlv_strct.CW.xManMode THEN
	EnableVlvAuto:= FALSE;
END_IF
Vlv_strct.SW.xManAuto:= EnableVlvAuto;
	
Vlv_strct.SW.xManOK:=NOT Vlv_strct.SW.xAlarmAccum AND Vlv_strct.CW.xAuxON AND Vlv_strct.CW.xEnable AND NOT EnableVlvAuto;
Vlv_strct.SW.xAutoOK:= NOT Vlv_strct.SW.xAlarmAccum AND Vlv_strct.CW.xAuxON AND Vlv_strct.CW.xEnable AND EnableVlvAuto AND Cycle.SW.xRunning;
	
	//Run in manual mode
IF Vlv_strct.CW.xManOpen OR Vlv_strct.CW.xManClose THEN
	Vlv_strct.SW.xRunManual:= TRUE;
END_IF
	
IF Vlv_strct.CW.xStop OR NOT IF Vlv_strct.CW.xStop OR NOT Vlv_strct.SW.xManOK THEN
	Vlv_strct.SW.xRunManual:= FALSE;
END_IF
	
	//Run in auto mode
Vlv_strct.SW.xRunAuto:= Cycle.SW.xRunning AND Vlv_strct.SW.xAutoOK;
	
	//Open/Close commands
COM_Open:= ((Vlv_strct.CW.xAutoOpen AND Vlv_strct.SW.xRunAuto AND Vlv_strct.SW.xAutoOK) OR ((Vlv_strct.CW.xManOpen OR COM_Open) AND Vlv_strct.SW.xRunManual AND Vlv_strct.SW.xManOK)) AND NOT COM_Close AND NOT Vlv_strct.SW.xOpened;
COM_Close:= ((Vlv_strct.CW.xAutoClose AND Vlv_strct.SW.xRunAuto AND Vlv_strct.SW.xAutoOK) OR ((Vlv_strct.CW.xManClose OR COM_Close) AND Vlv_strct.SW.xRunManual AND Vlv_strct.SW.xManOK)) AND NOT COM_Open AND NOT Vlv_strct.SW.xClosed;

IF Vlv_strct.CW.xSimEn THEN
	Vlv_strct.SW.xCOM_Open:= FALSE;
	Vlv_strct.SW.xCOM_Close:= FALSE;	
ELSE
	Vlv_strct.SW.xCOM_Open:= COM_Open;
	Vlv_strct.SW.xCOM_Close:= COM_Close;	
END_IF
	
	//Status processing
IF Vlv_strct.SW.xAlarmAccum  THEN
	Vlv_strct.wStatus:= VLV_Stat.ALARM_ACCUM;
ELSIF Vlv_strct.SW.xOpened THEN
	Vlv_strct.wStatus:= VLV_Stat.OPENED;
ELSIF Vlv_strct.SW.xClosed THEN
	Vlv_strct.wStatus:= VLV_Stat.CLOSED;
ELSIF NOT Vlv_strct.CW.xExtraEn THEN
	Vlv_strct.wStatus:= VLV_Stat.BLOCK;
ELSE
	Vlv_strct.wStatus:= VLV_Stat.STANDBY;
END_IF

	//Reset control bits
Vlv_strct.CW.xAutoMode:= FALSE;
Vlv_strct.CW.xManMode:= FALSE;
Vlv_strct.CW.xManOpen:= FALSE;
Vlv_strct.CW.xStop:= FALSE;
Vlv_strct.CW.xManClose:= FALSE;
Vlv_strct.CW.xACK:= FALSE;

          
END_FUNCTION_BLOCK

FUNCTION TimeNTPGet : DWORD
  VAR_IN_OUT
    pNtpServer_Addr : STRING;
    pResult : UDINT;
  END_VAR
  VAR
    tcpError : UDINT;
    socketHandle : RTS_IEC_HANDLE;
    socketAddress : SOCKADDRESS;
    sentBytes : DINT;
    receiveBuffer : ARRAY[1..64] OF BYTE;
    receivedBytes : DINT;
    sendbuf : ARRAY[1..48] OF BYTE := [16#DB, 47(0)];
    dwDateTime : DWORD;
    wRepeat : WORD := 0;
    secFrom1900to1970 : DWORD := 2208988800;  (* ////////// *)
  END_VAR

            IF pNtpServer_Addr='' THEN
	pNtpServer_Addr := '172.16.34.34';	

END_IF

socketHandle := SysSockCreate(SOCKET_AF_INET, SOCKET_DGRAM, SOCKET_IPPROTO_UDP, ADR(tcpError)); // SOCKET_DGRAM

IF TcpError =0 THEN 
        
   sendbuf[1]:=16#DB; //    NTP Client V3

// memset();
   socketAddress.sin_zero[0] := 0;
   socketAddress.sin_zero[1] := 0;
   socketAddress.sin_zero[2] := 0;
   socketAddress.sin_zero[3] := 0;
   socketAddress.sin_zero[4] := 0;
   socketAddress.sin_zero[5] := 0;
   socketAddress.sin_zero[6] := 0;
   socketAddress.sin_zero[7] := 0;
   socketAddress.sin_family:= SOCKET_AF_INET;
   socketAddress.sin_port:= SysSockHtons(123); // setting the port of the socket 37 - NTP

// Add to IP
   SysSockInetAddr(pNtpServer_Addr, ADR(socketAddress.sin_addr.ulAddr)); // setting the address of the socket     
   tcpError:= SysSockConnect(socketHandle, ADR(socketAddress), SIZEOF(socketAddress));
   IF TcpError =0 THEN 
      sentBytes:= SysSockSend(hSocket:= socketHandle, pbyBuffer:= ADR(sendbuf), diBufferSize:=SIZEOF(sendbuf), diFlags:= 0, pResult:= ADR(tcpError));
   END_IF
   IF TcpError =0 AND sentBytes = SIZEOF(sendbuf) THEN 
    REPEAT
		 receivedBytes:= SysSockGetRecvSizeUdp(hSocketUdp:= socketHandle, diTimeout :=0, pResult := ADR(tcpError));
		 IF receivedBytes=48 AND tcpError=0 THEN
           receivedBytes:= SysSockRecv(hSocket:= socketHandle, pbyBuffer:= ADR(receiveBuffer), diBufferSize:= SIZEOF(receiveBuffer), diFlags:= 0, pResult:= ADR(tcpError));		 
		 ELSE
  	        wRepeat := wRepeat+1;    
            sysTaskWaitSleep(0,1000);
         END_IF
         UNTIL (receivedBytes<>0 OR tcpError<>0) OR (wRepeat>=10)  // so wait 10 sec for very slow connection
      END_REPEAT;
   END_IF
   SysSockClose(socketHandle);
END_IF

pResult := tcpError;

IF receivedBytes <>48 OR pResult <> 0 THEN
    TimeNTPGet := 0;    //
	IF pResult = 0 THEN     // if we have no ethernet communication issue then use the timeout error code
		pResult := SEN.TimedOut;   // No valid response from NTP server
	END_IF
ELSE
	dwDateTime:=receiveBuffer[33];
    dwDateTime:=SHL(dwDateTime,8) + receiveBuffer[34];
    dwDateTime:=SHL(dwDateTime,8) + receiveBuffer[35];
    dwDateTime:=SHL(dwDateTime,8) + receiveBuffer[36];
    TimeNTPGet:= dwDateTime - secFrom1900to1970 + wRepeat;  // time correction for long response time
END_IF
          
END_FUNCTION

FUNCTION_BLOCK ReadNTPData
  VAR_INPUT
    xAuto : BOOL;
    xSync : BOOL;
    tSync : TIME;
    IP_addr : STRING;
    iBias : INT;
  END_VAR
  VAR_IN_OUT
    xPing : BOOL;
  END_VAR
  VAR
    dwLocalDateTime : DWORD;
    l_udiResult : UDINT;
    RtcTime : DWORD;
    fb_cycle : TON;
  END_VAR
  VAR_OUTPUT
    ServerDate : SysTimeRtc.SYSTIMEDATE;
    PLC_time : SysTimeRtc.SYSTIMEDATE;
    eError : UDINT := 0;
    xNTPSynchronously : BOOL := FALSE;
  END_VAR

            IF xAuto THEN
		fb_cycle(IN:=NOT fb_cycle.Q, PT:=tSync);
END_IF
IF fb_cycle.Q THEN
	xPing:=1;
END_IF
IF xPing THEN
dwLocalDateTime := TimeNTPGet(pNtpServer_Addr := IP_addr, pResult := eError);
IF eError = 0 THEN                   // if no error
	IF xSync THEN
		sysTimeRTCSet (dwLocalDateTime);
	END_IF
	SysTimeRtcConvertUtcToDate (dwTimestampUtc:=dwLocalDateTime,pDate:=ServerDate);
   xNTPSynchronously := TRUE;
ELSE
   xNTPSynchronously := FALSE; 
END_IF
END_IF

xPing := FALSE;   // event Get Time from NTP Server now completed 

RtcTime:=SysTimeRtcGet(pResult:=l_udiResult)+iBias*3600; 
SysTimeRtcConvertUtcToDate (dwTimestampUtc:=RtcTime,pDate:=PLC_time);
          
END_FUNCTION_BLOCK

PROGRAM prTimeManagment
  VAR
    uiResultGetTime : UDINT;
    stCurrentTimeDate : RTS_SYSTIMEDATE;
  END_VAR

(* CFC diagram, written out as Structured Text *)
SysTimeRtcConvertUtcToDate(SysTimeRtcGet(uiResultGetTime), stCurrentTimeDate);
wYear := stCurrentTimeDate;
wMonth := stCurrentTimeDate;
wDay := stCurrentTimeDate;
wHour := stCurrentTimeDate;
wMinute := stCurrentTimeDate;
wSecond := stCurrentTimeDate;
END_PROGRAM

PROGRAM Flow_meter
  VAR
    rFlwAccum_1 AT %MD20284 : REAL;
    rFlwAccum_2 AT %MD20285 : REAL;
    rFlwAccum_3 AT %MD20286 : REAL;
    rFlwAccum_4 AT %MD20287 : REAL;
    rFlwAccum_5 AT %MD20288 : REAL;
    rFlwAccum_6 AT %MD20289 : REAL;
    rFlwAccum_7 AT %MD20290 : REAL;
    rFlwAccum_8 AT %MD20291 : REAL;
    rFlwAccum_9 AT %MD20292 : REAL;
    rFlwAccum_10 AT %MD20293 : REAL;
    rFlwInst_1 AT %MD20276 : REAL;
    rFlwInst_2 AT %MD20277 : REAL;
    rFlwInst_3 AT %MD20278 : REAL;
    rFlwInst_4 AT %MD20279 : REAL;
    rFlwInst_5 AT %MD20280 : REAL;
    rFlwInst_6 AT %MD20281 : REAL;
  END_VAR
  VAR
    FB_ErrFlw_1 : Comm_error;
    FB_ErrFlw_2 : Comm_error;
    FB_ErrFlw_3 : Comm_error;
    FB_ErrFlw_4 : Comm_error;
    FB_ErrFlw_5 : Comm_error;
    FB_ErrFlw_6 : Comm_error;
    xErrFlw_1 : BOOL;
    xErrFlw_2 : BOOL;
    xErrFlw_3 : BOOL;
    xErrFlw_4 : BOOL;
    xErrFlw_5 : BOOL;
    xErrFlw_6 : BOOL;
  END_VAR

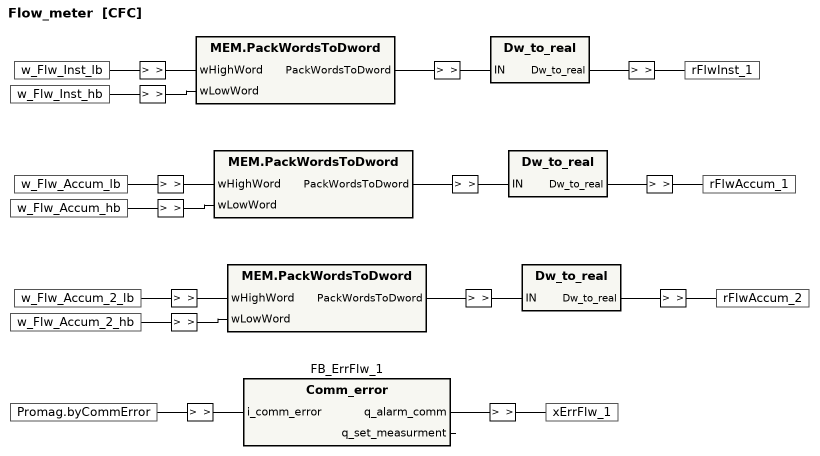
(* CFC diagram, written out as Structured Text *)
rFlwInst_1 := Dw_to_real(MEM.PackWordsToDword(w_Flw_Inst_lb, w_Flw_Inst_hb));
rFlwAccum_1 := Dw_to_real(MEM.PackWordsToDword(w_Flw_Accum_lb, w_Flw_Accum_hb));
rFlwAccum_2 := Dw_to_real(MEM.PackWordsToDword(w_Flw_Accum_2_lb, w_Flw_Accum_2_hb));
FB_ErrFlw_1(i_comm_error := Promag.byCommError);
xErrFlw_1 := FB_ErrFlw_1.q_alarm_comm;
END_PROGRAM

PROGRAM Power_meter
  VAR
    rVol12_1 AT %MD20086 : REAL;
    rVol23_1 AT %MD20096 : REAL;
    rVol31_1 AT %MD20106 : REAL;
    rVolAvg_1 AT %MD20116 : REAL;
    rCurA_1 AT %MD20046 : REAL;
    rCurB_1 AT %MD20056 : REAL;
    rCurC_1 AT %MD20066 : REAL;
    rCurAvg_1 AT %MD20076 : REAL;
    rTotPwrR_1 AT %MD20136 : REAL;  (* Мощность реактивная *)
    rTotPwrAp_1 AT %MD20146 : REAL;  (* apparent power полная мощность *)
    rPwrFact_1 AT %MD20156 : REAL;
    rCurFrq_1 AT %MD20166 : REAL;
    rEnergyA_1 AT %MD20176 : REAL;
    rEnergyR_1 AT %MD20186 : REAL;
    rTotPwrA_1 AT %MD20126 : REAL;  (* Мощность активная *)
    rCurA_2 AT %MD20047 : REAL;
    rCurB_2 AT %MD20057 : REAL;
    rCurC_2 AT %MD20067 : REAL;
    rCurAvg_2 AT %MD20077 : REAL;
    rVol12_2 AT %MD20087 : REAL;
    rVol23_2 AT %MD20097 : REAL;
    rVol31_2 AT %MD20107 : REAL;
    rVolAvg_2 AT %MD20117 : REAL;
    rTotPwrA_2 AT %MD20127 : REAL;
    rTotPwrR_2 AT %MD20137 : REAL;
    rTotPwrAp_2 AT %MD20147 : REAL;
    rPwrFact_2 AT %MD20157 : REAL;
    rCurFrq_2 AT %MD20167 : REAL;
    rEnergyA_2 AT %MD20177 : REAL;
    rEnergyR_2 AT %MD20187 : REAL;
    rCurA_3 AT %MD20048 : REAL;
    rCurA_4 AT %MD20049 : REAL;
    rCurA_5 AT %MD20050 : REAL;
    rCurA_6 AT %MD20051 : REAL;
    rCurA_7 AT %MD20052 : REAL;
    rCurA_8 AT %MD20053 : REAL;
    rCurA_9 AT %MD20054 : REAL;
    rCurA_10 AT %MD20055 : REAL;
    rCurB_3 AT %MD20058 : REAL;
    rCurB_4 AT %MD20059 : REAL;
    rCurB_5 AT %MD20060 : REAL;
    rCurB_6 AT %MD20061 : REAL;
    rCurB_7 AT %MD20062 : REAL;
    rCurB_8 AT %MD20063 : REAL;
    rCurB_9 AT %MD20064 : REAL;
    rCurB_10 AT %MD20065 : REAL;
    rCurC_3 AT %MD20068 : REAL;
    rCurC_4 AT %MD20069 : REAL;
    rCurC_5 AT %MD20070 : REAL;
    rCurC_6 AT %MD20071 : REAL;
    rCurC_7 AT %MD20072 : REAL;
    rCurC_8 AT %MD20073 : REAL;
    rCurC_9 AT %MD20074 : REAL;
    rCurC_10 AT %MD20075 : REAL;
    rCurAvg_3 AT %MD20078 : REAL;
    rCurAvg_4 AT %MD20079 : REAL;
    rCurAvg_5 AT %MD20080 : REAL;
    rCurAvg_6 AT %MD20081 : REAL;
    rCurAvg_7 AT %MD20082 : REAL;
    rCurAvg_8 AT %MD20083 : REAL;
    rCurAvg_9 AT %MD20084 : REAL;
    rCurAvg_10 AT %MD20085 : REAL;
    rVol12_3 AT %MD20088 : REAL;
    rVol12_4 AT %MD20089 : REAL;
    rVol12_5 AT %MD20090 : REAL;
    rVol12_6 AT %MD20091 : REAL;
    rVol12_7 AT %MD20092 : REAL;
    rVol12_8 AT %MD20093 : REAL;
    rVol12_9 AT %MD20094 : REAL;
    rVol12_10 AT %MD20095 : REAL;
    rVol23_3 AT %MD20098 : REAL;
    rVol23_4 AT %MD20099 : REAL;
    rVol23_5 AT %MD20100 : REAL;
    rVol23_6 AT %MD20101 : REAL;
    rVol23_7 AT %MD20102 : REAL;
    rVol23_8 AT %MD20103 : REAL;
    rVol23_9 AT %MD20104 : REAL;
    rVol23_10 AT %MD20105 : REAL;
    rVol31_3 AT %MD20108 : REAL;
    rVol31_4 AT %MD20109 : REAL;
    rVol31_5 AT %MD20110 : REAL;
    rVol31_6 AT %MD20111 : REAL;
    rVol31_7 AT %MD20112 : REAL;
    rVol31_8 AT %MD20113 : REAL;
    rVol31_9 AT %MD20114 : REAL;
    rVol31_10 AT %MD20115 : REAL;
    rVolAvg_3 AT %MD20118 : REAL;
    rVolAvg_4 AT %MD20119 : REAL;
    rVolAvg_5 AT %MD20120 : REAL;
    rVolAvg_6 AT %MD20121 : REAL;
    rVolAvg_7 AT %MD20122 : REAL;
    rVolAvg_8 AT %MD20123 : REAL;
    rVolAvg_9 AT %MD20124 : REAL;
    rVolAvg_10 AT %MD20125 : REAL;
    rTotPwrA_3 AT %MD20128 : REAL;
    rTotPwrA_4 AT %MD20129 : REAL;
    rTotPwrA_5 AT %MD20130 : REAL;
    rTotPwrA_6 AT %MD20131 : REAL;
    rTotPwrA_7 AT %MD20132 : REAL;
    rTotPwrA_8 AT %MD20133 : REAL;
    rTotPwrA_9 AT %MD20134 : REAL;
    rTotPwrA_10 AT %MD20135 : REAL;
    rTotPwrR_3 AT %MD20138 : REAL;
    rTotPwrR_4 AT %MD20139 : REAL;
    rTotPwrR_5 AT %MD20140 : REAL;
    rTotPwrR_6 AT %MD20141 : REAL;
    rTotPwrR_7 AT %MD20142 : REAL;
    rTotPwrR_8 AT %MD20143 : REAL;
    rTotPwrR_9 AT %MD20144 : REAL;
    rTotPwrR_10 AT %MD20145 : REAL;
    rTotPwrAp_3 AT %MD20148 : REAL;
    rTotPwrAp_4 AT %MD20149 : REAL;
    rTotPwrAp_5 AT %MD20150 : REAL;
    rTotPwrAp_6 AT %MD20151 : REAL;
    rTotPwrAp_7 AT %MD20152 : REAL;
    rTotPwrAp_8 AT %MD20153 : REAL;
    rTotPwrAp_9 AT %MD20154 : REAL;
    rTotPwrAp_10 AT %MD20155 : REAL;
    rPwrFact_3 AT %MD20158 : REAL;
    rPwrFact_4 AT %MD20159 : REAL;
    rPwrFact_5 AT %MD20160 : REAL;
    rPwrFact_6 AT %MD20161 : REAL;
    rPwrFact_7 AT %MD20162 : REAL;
    rPwrFact_8 AT %MD20163 : REAL;
    rPwrFact_9 AT %MD20164 : REAL;
    rPwrFact_10 AT %MD20165 : REAL;
    rCurFrq_3 AT %MD20168 : REAL;
    rCurFrq_4 AT %MD20169 : REAL;
    rCurFrq_5 AT %MD20170 : REAL;
    rCurFrq_6 AT %MD20171 : REAL;
    rCurFrq_7 AT %MD20172 : REAL;
    rCurFrq_8 AT %MD20173 : REAL;
    rCurFrq_9 AT %MD20174 : REAL;
    rCurFrq_10 AT %MD20175 : REAL;
    rEnergyA_3 AT %MD20178 : REAL;
    rEnergyA_4 AT %MD20179 : REAL;
    rEnergyA_5 AT %MD20180 : REAL;
    rEnergyA_6 AT %MD20181 : REAL;
    rEnergyA_7 AT %MD20182 : REAL;
    rEnergyA_8 AT %MD20183 : REAL;
    rEnergyA_9 AT %MD20184 : REAL;
    rEnergyA_10 AT %MD20185 : REAL;
    rEnergyA_11 AT %MD20186 : REAL;
    rEnergyA_12 AT %MD20187 : REAL;
    rEnergyA_13 AT %MD20188 : REAL;
    rEnergyA_14 AT %MD20189 : REAL;
    rEnergyR_3 AT %MD20188 : REAL;
    rEnergyR_4 AT %MD20189 : REAL;
    rEnergyR_5 AT %MD20190 : REAL;
    rEnergyR_6 AT %MD20191 : REAL;
    rEnergyR_7 AT %MD20192 : REAL;
    rEnergyR_8 AT %MD20193 : REAL;
    rEnergyR_9 AT %MD20194 : REAL;
    rEnergyR_10 AT %MD20195 : REAL;
    rEnergyR_11 AT %MD20196 : REAL;
    rEnergyR_12 AT %MD20197 : REAL;
    rEnergyR_13 AT %MD20198 : REAL;
    rEnergyR_14 AT %MD20199 : REAL;
    rEnergyA_1_L AT %MD20196 : DWORD;
    rEnergyA_1_H AT %MD20197 : DWORD;
    rEnergyR_1_L AT %MD20198 : DWORD;
    rEnergyR_1_H AT %MD20199 : DWORD;
    rEnergyA_2_L AT %MD20200 : DWORD;
    rEnergyA_2_H AT %MD20201 : DWORD;
    rEnergyR_2_L AT %MD20202 : DWORD;
    rEnergyR_2_H AT %MD20203 : DWORD;
    rEnergyA_3_L AT %MD20204 : DWORD;
    rEnergyA_3_H AT %MD20205 : DWORD;
    rEnergyR_3_L AT %MD20206 : DWORD;
    rEnergyR_3_H AT %MD20207 : DWORD;
    rEnergyA_4_L AT %MD20208 : DWORD;
    rEnergyA_4_H AT %MD20209 : DWORD;
    rEnergyR_4_L AT %MD20210 : DWORD;
    rEnergyR_4_H AT %MD20211 : DWORD;
    rEnergyA_5_L AT %MD20212 : DWORD;
    rEnergyA_5_H AT %MD20213 : DWORD;
    rEnergyR_5_L AT %MD20214 : DWORD;
    rEnergyR_5_H AT %MD20215 : DWORD;
    rEnergyA_6_L AT %MD20216 : DWORD;
    rEnergyA_6_H AT %MD20217 : DWORD;
    rEnergyR_6_L AT %MD20218 : DWORD;
    rEnergyR_6_H AT %MD20219 : DWORD;
    rEnergyA_7_L AT %MD20220 : DWORD;
    rEnergyA_7_H AT %MD20221 : DWORD;
    rEnergyR_7_L AT %MD20222 : DWORD;
    rEnergyR_7_H AT %MD20223 : DWORD;
    rEnergyA_8_L AT %MD20224 : DWORD;
    rEnergyA_8_H AT %MD20225 : DWORD;
    rEnergyR_8_L AT %MD20226 : DWORD;
    rEnergyR_8_H AT %MD20227 : DWORD;
    rEnergyA_9_L AT %MD20228 : DWORD;
    rEnergyA_9_H AT %MD20229 : DWORD;
    rEnergyR_9_L AT %MD20230 : DWORD;
    rEnergyR_9_H AT %MD20231 : DWORD;
    rEnergyA_10_L AT %MD20232 : DWORD;
    rEnergyA_10_H AT %MD20233 : DWORD;
    rEnergyR_10_L AT %MD20234 : DWORD;
    rEnergyR_10_H AT %MD20235 : DWORD;
    rCurA_11 AT %MD20300 : REAL;
    rCurB_11 AT %MD20301 : REAL;
    rCurC_11 AT %MD20302 : REAL;
    rCurAvg_11 AT %MD20303 : REAL;
    rVol12_11 AT %MD20304 : REAL;
    rVol23_11 AT %MD20305 : REAL;
    rVol31_11 AT %MD20306 : REAL;
    rVolAvg_11 AT %MD20307 : REAL;
    rTotPwrA_11 AT %MD20308 : REAL;
    rTotPwrR_11 AT %MD20309 : REAL;
    rTotPwrAp_11 AT %MD20310 : REAL;
    rPwrFact_11 AT %MD20311 : REAL;
    rCurFrq_11 AT %MD20312 : REAL;
    rEnergyA_11_L AT %MD20313 : DWORD;
    rEnergyA_11_H AT %MD20314 : DWORD;
    rEnergyR_11_L AT %MD20315 : DWORD;
    rEnergyR_11_H AT %MD20316 : DWORD;
    RcurA_12 AT %MD20317 : REAL;
    rCurB_12 AT %MD20318 : REAL;
    rCurC_12 AT %MD20319 : REAL;
    rCurAvg_12 AT %MD20320 : REAL;
    rVol12_12 AT %MD20321 : REAL;
    rVol23_12 AT %MD20322 : REAL;
    rVol31_12 AT %MD20323 : REAL;
    rVolAvg_12 AT %MD20324 : REAL;
    rTotPwrA_12 AT %MD20325 : REAL;
    rTotPwrR_12 AT %MD20326 : REAL;
    rTotPwrAp_12 AT %MD20327 : REAL;
    rPwrFact_12 AT %MD20328 : REAL;
    rCurFrq_12 AT %MD20329 : REAL;
    rEnergyA_12_L AT %MD20330 : DWORD;
    rEnergyA_12_H AT %MD20331 : DWORD;
    rEnergyR_12_L AT %MD20332 : DWORD;
    rEnergyR_12_H AT %MD20333 : DWORD;
    RcurA_13 AT %MD20334 : REAL;
    rCurB_13 AT %MD20335 : REAL;
    rCurC_13 AT %MD20336 : REAL;
    rCurAvg_13 AT %MD20337 : REAL;
    rVol12_13 AT %MD20338 : REAL;
    rVol23_13 AT %MD20339 : REAL;
    rVol31_13 AT %MD20340 : REAL;
    rVolAvg_13 AT %MD20341 : REAL;
    rTotPwrA_13 AT %MD20342 : REAL;
    rTotPwrR_13 AT %MD20343 : REAL;
    rTotPwrAp_13 AT %MD20344 : REAL;
    rPwrFact_13 AT %MD20345 : REAL;
    rCurFrq_13 AT %MD20346 : REAL;
    rEnergyA_13_L AT %MD20347 : DWORD;
    rEnergyA_13_H AT %MD20348 : DWORD;
    rEnergyR_13_L AT %MD20349 : DWORD;
    rEnergyR_13_H AT %MD20350 : DWORD;
    RcurA_14 AT %MD20351 : REAL;
    rCurB_14 AT %MD20352 : REAL;
    rCurC_14 AT %MD20353 : REAL;
    rCurAvg_14 AT %MD20354 : REAL;
    rVol12_14 AT %MD20355 : REAL;
    rVol23_14 AT %MD20356 : REAL;
    rVol31_14 AT %MD20357 : REAL;
    rVolAvg_14 AT %MD20358 : REAL;
    rTotPwrA_14 AT %MD20359 : REAL;
    rTotPwrR_14 AT %MD20360 : REAL;
    rTotPwrAp_14 AT %MD20361 : REAL;
    rPwrFact_14 AT %MD20362 : REAL;
    rCurFrq_14 AT %MD20363 : REAL;
    rEnergyA_14_L AT %MD20364 : DWORD;
    rEnergyA_14_H AT %MD20365 : DWORD;
    rEnergyR_14_L AT %MD20366 : DWORD;
    rEnergyR_14_H AT %MD20367 : DWORD;
  END_VAR
  VAR
    pm_1 : Power_c;
    pm_2 : Power_c;
    pm_3 : Power_c;
    pm_4 : Power_c;
    pm_5 : Power_c;
    pm_6 : Power_c;
    pm_7 : Power_c;
    pm_8 : Power_c;
    pm_9 : Power_c;
    pm_10 : Power_c;
    pm_11 : Power_c;
    pm_12 : Power_c;
    pm_13 : Power_c;
    pm_14 : Power_c;
    xErrPwrMtr_1 : BOOL;
    xErrPwrMtr_2 : BOOL;
    xErrPwrMtr_3 : BOOL;
    xErrPwrMtr_4 : BOOL;
    xErrPwrMtr_5 : BOOL;
    xErrPwrMtr_6 : BOOL;
    xErrPwrMtr_7 : BOOL;
    xErrPwrMtr_8 : BOOL;
    xErrPwrMtr_9 : BOOL;
    xErrPwrMtr_10 : BOOL;
    xErrPwrMtr_11 : BOOL;
    xErrPwrMtr_12 : BOOL;
    xErrPwrMtr_13 : BOOL;
    xErrPwrMtr_14 : BOOL;
  END_VAR

            pm_1( //Counter №1
	PM_FB:= PM325x_Modbus_Slave_FB, 
	com_err:= PM325x_Modbus_Slave.byCommError, 
	modbus_slave_ch6:= ADR(iwPM325x_Modbus_Slave_Channel_6),
	x_alarm_comm=>xErrPwrMtr_1, 	
	rCurA=>rCurA_1, rCurB=> rCurB_1, rCurC=>rCurC_1, rCurAvg=>rCurAvg_1, 
	rVol12=>rVol12_1, rVol23=>rVol23_1, rVol31=>rVol31_1, rVolAvg=>rVolAvg_1 , 
	rTotPwrA=>rTotPwrA_1, rTotPwrR=>rTotPwrR_1, rTotPwrAp=>rTotPwrAp_1 , 
	rPwrFact=>rPwrFact_1, rCurFrq=>rCurFrq_1, rEnergyA=> rEnergyA_1, rEnergyR=>rEnergyR_1,
	rEnergyA_L=>rEnergyA_1_L, rEnergyA_H=>rEnergyA_1_H, rEnergyR_L=>rEnergyR_1_L, rEnergyR_H=>rEnergyR_1_H );
	
pm_2( //Counter №2
	PM_FB:= PM325x_Modbus_Slave_1_FB, 
	com_err:= PM325x_Modbus_Slave_1.byCommError, 
	modbus_slave_ch6:= ADR(iwPM325x_Modbus_Slave_1_Channel_6),
	x_alarm_comm=>xErrPwrMtr_2, 	
	rCurA=>rCurA_2, rCurB=>rCurB_2, rCurC=>rCurC_2, rCurAvg=>rCurAvg_2, 
	rVol12=>rVol12_2, rVol23=>rVol23_2 , rVol31=>rVol31_2, rVolAvg=>rVolAvg_2 , 
	rTotPwrA=>rTotPwrA_2, rTotPwrR=>rTotPwrR_2, rTotPwrAp=>rTotPwrAp_2 , 
	rPwrFact=>rPwrFact_2, rCurFrq=>rCurFrq_2, rEnergyA=>rEnergyA_2, rEnergyR=>rEnergyR_2,
	rEnergyA_L=>rEnergyA_2_L, rEnergyA_H=>rEnergyA_2_H, rEnergyR_L=>rEnergyR_2_L, rEnergyR_H=>rEnergyR_2_H );
(*
pm_3( //Counter №3
	PM_FB:= PM325x_Modbus_Slave_2_FB, 
	com_err:= PM325x_Modbus_Slave_2.byCommError, 
	modbus_slave_ch6:= ADR(iwPM325x_Modbus_Slave_2_Channel_6),
	x_alarm_comm=>xErrPwrMtr_3, 	
	rCurA=>rCurA_3, rCurB=>rCurB_3, rCurC=> rCurC_3, rCurAvg=>rCurAvg_3, 
	rVol12=>rVol12_3, rVol23=>rVol23_3, rVol31=>rVol31_3, rVolAvg=>rVolAvg_3 , 
	rTotPwrA=>rTotPwrA_3, rTotPwrR=>rTotPwrR_3, rTotPwrAp=>rTotPwrAp_3 , 
	rPwrFact=>rPwrFact_3, rCurFrq=>rCurFrq_3, rEnergyA=>rEnergyA_3, rEnergyR=>rEnergyR_3,
	rEnergyA_L=>rEnergyA_3_L, rEnergyA_H=>rEnergyA_3_H, rEnergyR_L=>rEnergyR_3_L, rEnergyR_H=>rEnergyR_3_H );

pm_4( //Counter №4
	PM_FB:= PM325x_Modbus_Slave_3_FB, 
	com_err:= PM325x_Modbus_Slave_3.byCommError, 
	modbus_slave_ch6:= ADR(iwPM325x_Modbus_Slave_3_Channel_6),
	x_alarm_comm=>xErrPwrMtr_4, 	
	rCurA=>rCurA_4, rCurB=>rCurB_4, rCurC=>rCurC_4, rCurAvg=> rCurAvg_4, 
	rVol12=>rVol12_4, rVol23=>rVol23_4, rVol31=>rVol31_4, rVolAvg=>rVolAvg_4 , 
	rTotPwrA=>rTotPwrA_4, rTotPwrR=>rTotPwrR_4, rTotPwrAp=>rTotPwrAp_4 , 
	rPwrFact=>rPwrFact_4, rCurFrq=>rCurFrq_4, rEnergyA=>rEnergyA_4, rEnergyR=>rEnergyR_4,
	rEnergyA_L=>rEnergyA_4_L, rEnergyA_H=>rEnergyA_4_H, rEnergyR_L=>rEnergyR_4_L, rEnergyR_H=>rEnergyR_4_H );

pm_5( //Counter №5
	PM_FB:= PM325x_Modbus_Slave_4_FB, 
	com_err:= PM325x_Modbus_Slave_4.byCommError, 
	modbus_slave_ch6:= ADR(iwPM325x_Modbus_Slave_4_Channel_6),
	x_alarm_comm=>xErrPwrMtr_5, 	
	rCurA=>rCurA_5, rCurB=>rCurB_5, rCurC=>rCurC_5, rCurAvg=>rCurAvg_5, 
	rVol12=>rVol12_5, rVol23=>rVol23_5, rVol31=>rVol31_5, rVolAvg=>rVolAvg_5 , 
	rTotPwrA=>rTotPwrA_5, rTotPwrR=>rTotPwrR_5, rTotPwrAp=>rTotPwrAp_5 , 
	rPwrFact=>rPwrFact_5, rCurFrq=>rCurFrq_5, rEnergyA=>rEnergyA_5, rEnergyR=>rEnergyR_5,
	rEnergyA_L=>rEnergyA_5_L, rEnergyA_H=>rEnergyA_5_H, rEnergyR_L=>rEnergyR_5_L, rEnergyR_H=>rEnergyR_5_H );

pm_6( //Counter №6
	PM_FB:= PM325x_Modbus_Slave_5_FB, 
	com_err:= PM325x_Modbus_Slave_5.byCommError, 
	modbus_slave_ch6:= ADR(iwPM325x_Modbus_Slave_5_Channel_6),
	x_alarm_comm=>xErrPwrMtr_6, 	
	rCurA=> rCurA_6, rCurB=>rCurB_6, rCurC=>rCurC_6, rCurAvg=> rCurAvg_6, 
	rVol12=>rVol12_6, rVol23=>rVol23_6, rVol31=>rVol31_6, rVolAvg=>rVolAvg_6 , 
	rTotPwrA=> rTotPwrA_6, rTotPwrR=>rTotPwrR_6, rTotPwrAp=>rTotPwrAp_6 , 
	rPwrFact=> rPwrFact_6, rCurFrq=>rCurFrq_6, rEnergyA=>rEnergyA_6, rEnergyR=>rEnergyR_6,
	rEnergyA_L=>rEnergyA_6_L, rEnergyA_H=>rEnergyA_6_H, rEnergyR_L=>rEnergyR_6_L, rEnergyR_H=>rEnergyR_6_H );
	
pm_7( //Counter №7
	PM_FB:= PM325x_Modbus_Slave_6_FB, 
	com_err:= PM325x_Modbus_Slave_6.byCommError, 
	modbus_slave_ch6:= ADR(iwPM325x_Modbus_Slave_6_Channel_6),
	x_alarm_comm=>xErrPwrMtr_7, 	
	rCurA=>rCurA_7, rCurB=>rCurB_7, rCurC=>rCurC_7, rCurAvg=> rCurAvg_7, 
	rVol12=>rVol12_7, rVol23=>rVol23_7, rVol31=>rVol31_7, rVolAvg=>rVolAvg_7 , 
	rTotPwrA=>rTotPwrA_7, rTotPwrR=>rTotPwrR_7, rTotPwrAp=>rTotPwrAp_7 , 
	rPwrFact=>rPwrFact_7, rCurFrq=>rCurFrq_7, rEnergyA=>rEnergyA_7, rEnergyR=>rEnergyR_7,
	rEnergyA_L=>rEnergyA_7_L, rEnergyA_H=>rEnergyA_7_H, rEnergyR_L=>rEnergyR_7_L, rEnergyR_H=>rEnergyR_7_H );

pm_8( //Counter №8
	PM_FB:= PM325x_Modbus_Slave_7_FB, 
	com_err:= PM325x_Modbus_Slave_7.byCommError, 
	modbus_slave_ch6:= ADR(iwPM325x_Modbus_Slave_7_Channel_6),
	x_alarm_comm=>xErrPwrMtr_8, 	
	rCurA=>rCurA_8, rCurB=>rCurB_8, rCurC=>rCurC_8, rCurAvg=>rCurAvg_8, 
	rVol12=>rVol12_8, rVol23=>rVol23_8, rVol31=>rVol31_8 ,rVolAvg=>rVolAvg_8 , 
	rTotPwrA=>rTotPwrA_8, rTotPwrR=>rTotPwrR_8, rTotPwrAp=>rTotPwrAp_8 , 
	rPwrFact=>rPwrFact_8, rCurFrq=>rCurFrq_8, rEnergyA=>rEnergyA_8, rEnergyR=>rEnergyR_8,
	rEnergyA_L=>rEnergyA_8_L, rEnergyA_H=>rEnergyA_8_H, rEnergyR_L=>rEnergyR_8_L, rEnergyR_H=>rEnergyR_8_H );

pm_9( //Counter №9
	PM_FB:= PM325x_Modbus_Slave_8_FB, 
	com_err:= PM325x_Modbus_Slave_8.byCommError, 
	modbus_slave_ch6:= ADR(iwPM325x_Modbus_Slave_8_Channel_6),
	x_alarm_comm=>xErrPwrMtr_9, 	
	rCurA=>rCurA_9, rCurB=>rCurB_9, rCurC=>rCurC_9, rCurAvg=>rCurAvg_9, 
	rVol12=>rVol12_9, rVol23=>rVol23_9 , rVol31=>rVol31_9, rVolAvg=>rVolAvg_9 , 
	rTotPwrA=>rTotPwrA_9, rTotPwrR=>rTotPwrR_9, rTotPwrAp=>rTotPwrAp_9 , 
	rPwrFact=>rPwrFact_9, rCurFrq=>rCurFrq_9, rEnergyA=>rEnergyA_9, rEnergyR=>rEnergyR_9,
	rEnergyA_L=>rEnergyA_9_L, rEnergyA_H=>rEnergyA_9_H, rEnergyR_L=>rEnergyR_9_L, rEnergyR_H=>rEnergyR_9_H );
	
pm_10( //Counter №10
	PM_FB:= PM325x_Modbus_Slave_9_FB, 
	com_err:= PM325x_Modbus_Slave_9.byCommError, 
	modbus_slave_ch6:= ADR(iwPM325x_Modbus_Slave_9_Channel_6),
	x_alarm_comm=>xErrPwrMtr_10, 	
	rCurA=>rCurA_10, rCurB=>rCurB_10, rCurC=>rCurC_10, rCurAvg=>rCurAvg_10, 
	rVol12=>rVol12_10, rVol23=>rVol23_10, rVol31=>rVol31_10, rVolAvg=>rVolAvg_10 , 
	rTotPwrA=>rTotPwrA_10, rTotPwrR=>rTotPwrR_10, rTotPwrAp=>rTotPwrAp_10 , 
	rPwrFact=>rPwrFact_10, rCurFrq=>rCurFrq_10, rEnergyA=>rEnergyA_10, rEnergyR=>rEnergyR_10,
	rEnergyA_L=>rEnergyA_10_L, rEnergyA_H=>rEnergyA_10_H, rEnergyR_L=>rEnergyR_10_L, rEnergyR_H=>rEnergyR_10_H );
	
pm_11( //Counter №11
	PM_FB:= PM325x_Modbus_Slave_10_FB, 
	com_err:= PM325x_Modbus_Slave_10.byCommError, 
	modbus_slave_ch6:= ADR(iwPM325x_Modbus_Slave_10_Channel_6),
	x_alarm_comm=>xErrPwrMtr_11, 	
	rCurA=>rCurA_11, rCurB=>rCurB_11, rCurC=>rCurC_11, rCurAvg=>rCurAvg_11, 
	rVol12=>rVol12_11, rVol23=>rVol23_11, rVol31=>rVol31_11, rVolAvg=>rVolAvg_11 , 
	rTotPwrA=>rTotPwrA_11, rTotPwrR=>rTotPwrR_11, rTotPwrAp=>rTotPwrAp_11 , 
	rPwrFact=>rPwrFact_11, rCurFrq=>rCurFrq_11, rEnergyA=>rEnergyA_11, rEnergyR=>rEnergyR_11,
	rEnergyA_L=>rEnergyA_11_L, rEnergyA_H=>rEnergyA_11_H, rEnergyR_L=>rEnergyR_11_L, rEnergyR_H=>rEnergyR_11_H );
	
pm_12( //Counter №12
	PM_FB:= PM325x_Modbus_Slave_11_FB, 
	com_err:= PM325x_Modbus_Slave_11.byCommError, 
	modbus_slave_ch6:= ADR(iwPM325x_Modbus_Slave_11_Channel_6),
	x_alarm_comm=>xErrPwrMtr_12, 	
	rCurA=>rCurA_12, rCurB=>rCurB_12, rCurC=>rCurC_12, rCurAvg=>rCurAvg_12, 
	rVol12=>rVol12_12, rVol23=>rVol23_12, rVol31=>rVol31_12, rVolAvg=>rVolAvg_12 , 
	rTotPwrA=>rTotPwrA_12, rTotPwrR=>rTotPwrR_12, rTotPwrAp=>rTotPwrAp_12 , 
	rPwrFact=>rPwrFact_12, rCurFrq=>rCurFrq_12, rEnergyA=>rEnergyA_12, rEnergyR=>rEnergyR_12,
	rEnergyA_L=>rEnergyA_12_L, rEnergyA_H=>rEnergyA_12_H, rEnergyR_L=>rEnergyR_12_L, rEnergyR_H=>rEnergyR_12_H );
	
pm_13( //Counter №13
	PM_FB:= PM325x_Modbus_Slave_12_FB, 
	com_err:= PM325x_Modbus_Slave_12.byCommError, 
	modbus_slave_ch6:= ADR(iwPM325x_Modbus_Slave_12_Channel_6),
	x_alarm_comm=>xErrPwrMtr_13, 	
	rCurA=>rCurA_13, rCurB=>rCurB_13, rCurC=>rCurC_13, rCurAvg=>rCurAvg_13, 
	rVol12=>rVol12_13, rVol23=>rVol23_13, rVol31=>rVol31_13, rVolAvg=>rVolAvg_13 , 
	rTotPwrA=>rTotPwrA_13, rTotPwrR=>rTotPwrR_13, rTotPwrAp=> rTotPwrAp_13 , 
	rPwrFact=>rPwrFact_13, rCurFrq=>rCurFrq_13, rEnergyA=>rEnergyA_13, rEnergyR=>rEnergyR_13,
	rEnergyA_L=>rEnergyA_13_L, rEnergyA_H=>rEnergyA_13_H, rEnergyR_L=>rEnergyR_13_L, rEnergyR_H=>rEnergyR_13_H );
	
pm_14( //Counter №14
	PM_FB:= PM325x_Modbus_Slave_13_FB, 
	com_err:= PM325x_Modbus_Slave_13.byCommError, 
	modbus_slave_ch6:= ADR(iwPM325x_Modbus_Slave_13_Channel_6),
	x_alarm_comm=>xErrPwrMtr_14, 	
	rCurA=>rCurA_14, rCurB=> rCurB_14, rCurC=>rCurC_14, rCurAvg=>rCurAvg_14, 
	rVol12=>rVol12_14, rVol23=>rVol23_14, rVol31=>rVol31_14, rVolAvg=>rVolAvg_14 , 
	rTotPwrA=>rTotPwrA_14, rTotPwrR=>rTotPwrR_14, rTotPwrAp=>rTotPwrAp_14 , 
	rPwrFact=>rPwrFact_14, rCurFrq=>rCurFrq_14, rEnergyA=>rEnergyA_14, rEnergyR=>rEnergyR_14,
	rEnergyA_L=>rEnergyA_14_L, rEnergyA_H=>rEnergyA_14_H, rEnergyR_L=>rEnergyR_14_L, rEnergyR_H=>rEnergyR_14_H );
*)	
(*pm_15( //Counter №15
	PM_FB:= PM325x_Modbus_Slave_1_FB, 
	com_err:= PM325x_Modbus_Slave_1.byCommError, 
	modbus_slave_ch6:= ADR(iwPM325x_Modbus_Slave_1_Channel_6),
	x_alarm_comm=>xErrPwrMtr_15, 	
	rCurA=>rCurA_15, rCurB=>rCurB_15, rCurC=>rCurC_15, rCurAvg=>rCurAvg_15, 
	rVol12=>rVol12_15, rVol23=>rVol23_15 , rVol31=>rVol31_15, rVolAvg=>rVolAvg_15 , 
	rTotPwrA=>rTotPwrA_15, rTotPwrR=>rTotPwrR_15, rTotPwrAp=>rTotPwrAp_15 , 
	rPwrFact=>rPwrFact_15, rCurFrq=>rCurFrq_15, rEnergyA=>rEnergyA_15, rEnergyR=>rEnergyR_15 );*)
          
END_PROGRAM

PROGRAM SP_control
  VAR
    wCmdSP AT %MW41005 : WORD;
    wNumSP AT %MW41606 : WORD;
    rPrsDN AT %MD20297 : REAL;
    rPrsSched AT %MD20296 : REAL;
    rSP_manual AT %MD20298 : REAL;
    wPrsHourSP_1 AT %MW41610 : WORD := 6;
    wPrsMinSP_1 AT %MW41611 : WORD := 30;
    wPrsMinSP_2 AT %MW41613 : WORD := 22;
    wPrsHourSP_2 AT %MW41612 : WORD := 0;
    wPrsHourSP_3 AT %MW41614 : WORD := 6;
    wPrsMinSP_3 AT %MW41615 : WORD := 45;
    wPrsMinSP_4 AT %MW41617 : WORD := 30;
    wPrsHourSP_4 AT %MW41616 : WORD := 21;
    wPrsMonthS AT %MW41619 : WORD := 5;
    wPrsDayS AT %MW41618 : WORD := 1;
    wPrsMonthW AT %MW41621 : WORD := 10;
    wPrsDayW AT %MW41620 : WORD := 10;
    wPrsHourSP_N AT %MW41622 : WORD;
    wPrsMinSP_N AT %MW41623 : WORD;
    r_SP_Current AT %MD20299 : REAL;
  END_VAR
  VAR
    Comm : BOOL;
    timer_res : TON;
    smmr : BOOL;
    setpoint : WORD;
    timer_comm : TON;
    rs_comm : RS;
    target : REAL;
    derv : DERIVATIVE;
    sp_wr : BOOL;
    rs_wr : RS;
    timer_wr : TON;
  END_VAR
  VAR_OUTPUT
    rPrsSP_1 AT %MD20292 : REAL;
    rPrsSP_2 AT %MD20293 : REAL;
    rPrsSP_3 AT %MD20294 : REAL;
    rPrsSP_4 AT %MD20295 : REAL;
  END_VAR
  VAR  (* added by the conversion: wires and edge detectors of the diagram *)
    _SP_change1_wPrsMinSP_1 : ANY;
    _SP_change1_wPrsHourSP_2 : ANY;
    _SP_change1_wPrsMinSP_2 : ANY;
    _SP_change1_wPrsHourSP_3 : ANY;
    _SP_change1_wPrsMinSP_3 : ANY;
    _SP_change1_wPrsHourSP_4 : ANY;
    _SP_change1_wPrsMinSP_4 : ANY;
    _SP_change1_Summer : ANY;
    _SP_change1_rPrsSP_1 : ANY;
    _SP_change1_rPrsSP_2 : ANY;
    _SP_change1_rPrsSP_3 : ANY;
    _SP_change1_rPrsSP_4 : ANY;
    _SP_change1_SP_target : ANY;
    _SP_change1_SP : ANY;
    _SP_change1_OUT : WORD;
  END_VAR

(* CFC diagram, written out as Structured Text *)
timer_res(IN := wCmdSP.2, PT := t#60s);
IF timer_res.Q THEN wCmdSP.2 := FALSE; END_IF;
timer_comm(IN := NOT wCmdSP.2, PT := t#60s);
rs_comm(SET := wCmdSP.2, RESET1 := timer_comm.Q);
_SP_change1_OUT := SP_change(wNumSP := wNumSP, rPrsDN := rPrsDN, rPrsSched := rPrsSched, rSP_manual := rSP_manual, wPrsHourSP_N := wPrsHourSP_N, wPrsMinSP_N := wPrsMinSP_N, xSCADA_Comm := rs_comm.Q1, r_dSP := 0.5, wPrsDayS := wPrsDayS, wPrsMonthS := wPrsMonthS, wPrsDayW := wPrsDayW, wPrsMonthW := wPrsMonthW, wCmdSP := wCmdSP, wPrsMinSP_1 => _SP_change1_wPrsMinSP_1, wPrsHourSP_2 => _SP_change1_wPrsHourSP_2, wPrsMinSP_2 => _SP_change1_wPrsMinSP_2, wPrsHourSP_3 => _SP_change1_wPrsHourSP_3, wPrsMinSP_3 => _SP_change1_wPrsMinSP_3, wPrsHourSP_4 => _SP_change1_wPrsHourSP_4, wPrsMinSP_4 => _SP_change1_wPrsMinSP_4, Summer => _SP_change1_Summer, rPrsSP_1 => _SP_change1_rPrsSP_1, rPrsSP_2 => _SP_change1_rPrsSP_2, rPrsSP_3 => _SP_change1_rPrsSP_3, rPrsSP_4 => _SP_change1_rPrsSP_4, SP_target => _SP_change1_SP_target, SP => _SP_change1_SP);
wPrsHourSP_1 := _SP_change1_OUT;
wPrsMinSP_1 := _SP_change1_wPrsMinSP_1;
wPrsHourSP_2 := _SP_change1_wPrsHourSP_2;
derv(IN := _SP_change1_SP, TM := 200);
wPrsMinSP_2 := _SP_change1_wPrsMinSP_2;
wPrsHourSP_3 := _SP_change1_wPrsHourSP_3;
wPrsMinSP_3 := _SP_change1_wPrsMinSP_3;
wPrsHourSP_4 := _SP_change1_wPrsHourSP_4;
setpoint := REAL_TO_WORD(_SP_change1_SP * 10);
wPrsMinSP_4 := _SP_change1_wPrsMinSP_4;
smmr := _SP_change1_Summer;
rPrsSP_1 := _SP_change1_rPrsSP_1;
rPrsSP_2 := _SP_change1_rPrsSP_2;
rPrsSP_3 := _SP_change1_rPrsSP_3;
rPrsSP_4 := _SP_change1_rPrsSP_4;
target := _SP_change1_SP_target;
sp_wr := <>(derv.OUT, 0);
r_SP_Current := _SP_change1_SP;
END_PROGRAM

PROGRAM Set_IP_Address
  VAR
    i_input_Mask_ip AT %MB250 : ARRAY[1..4] OF BYTE;
  END_VAR
  VAR
    i_input_Gateway_ip : ARRAY[1..4] OF BYTE;
  END_VAR

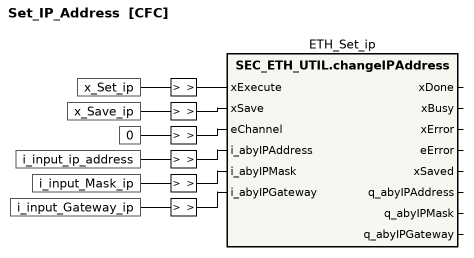
(* CFC diagram, written out as Structured Text *)
ETH_Set_ip(xExecute := x_Set_ip, xSave := x_Save_ip, eChannel := 0, i_abyIPAddress := i_input_ip_address, i_abyIPMask := i_input_Mask_ip, i_abyIPGateway := i_input_Gateway_ip);
END_PROGRAM

PROGRAM Alarm
  VAR
    wErrTmp_1 AT %MW41002 : WORD;
    wErrTmp_2 AT %MW41003 : WORD;
    wErrPrs AT %MW41001 : WORD;
    wErrLvl AT %MW41008 : WORD;
    wErrFlw AT %MW41000 : WORD;
    wErrPwrMtr AT %MW41006 : WORD;
    wErrOthr AT %MW41004 : WORD;
  END_VAR
  VAR
    fb_wErrTmp_1 : BIT_AS_WORD;
    fb_wErrTmp_2 : BIT_AS_WORD;
    fb_wErrPrs : BIT_AS_WORD;
    fb_wErrLvl : BIT_AS_WORD;
    fb_wErrFlw : BIT_AS_WORD;
    fb_ErrPwrMtr : BIT_AS_WORD;
    fb_errothr : BIT_AS_WORD;
    xErrorAccum : BOOL;
  END_VAR

            fb_wErrTmp_1(		//T sensor errors
	B00:= AI.xErrTmp_1, B01:= AI.xErrTmp_2, B02:= AI.xErrTmp_3, B03:= AI.xErrTmp_4, 
	B04:= AI.xErrTmp_5, B05:= AI.xErrTmp_6, B06:= AI.xErrTmp_7, B07:= AI.xErrTmp_8, 
	B08:= AI.xErrTmp_9, B09:= AI.xErrTmp_10, B10:= AI.xErrTmp_11, B11:= AI.xErrTmp_12, 
	B12:= AI.xErrTmp_13, B13:= AI.xErrTmp_14, B14:= AI.xErrTmp_5, B15:= AI.xErrTmp_16, 
W=> wErrTmp_1);
fb_wErrTmp_2(		//T sensor errors
	B00:= AI.xErrTmp_17, B01:= AI.xErrTmp_18, B02:= AI.xErrTmp_19, B03:= AI.xErrTmp_20, 
	B04:= AI.xErrTmp_21, B05:= AI.xErrTmp_22, B06:= AI.xErrTmp_23, B07:= AI.xErrTmp_24, 
	B08:= AI.xErrTmp_25, B09:= AI.xErrTmp_26, B10:= AI.xErrTmp_27, B11:= AI.xErrTmp_28, 
	B12:= AI.xErrTmp_29, B13:= AI.xErrTmp_30,
W=> wErrTmp_2);

fb_wErrPrs(			//P sensor errors
	B00:= AI.xErrPrs_1, B01:= AI.xErrPrs_2, B02:= AI.xErrPrs_3, 
	B03:= AI.xErrPrs_4, B04:= AI.xErrPrs_5, B05:= AI.xErrPrs_6, 
W=> wErrPrs);

fb_wErrLvl(			//L sensor errors
	B00:= AI.xErrLvl_1, B01:= AI.xErrLvl_2, B02:= AI.xErrLvl_3, 
	B03:= AI.xErrLvl_4, B04:= AI.xErrLvl_5, B05:= AI.xErrLvl_6, 
W=> wErrLvl);

fb_wErrFlw(			//F sensor errors
	B00:= Flow_meter.xErrFlw_1, B01:= Flow_meter.xErrFlw_2, B02:= Flow_meter.xErrFlw_3, 
	B03:= Flow_meter.xErrFlw_4, B04:= Flow_meter.xErrFlw_5, B05:= Flow_meter.xErrFlw_6, 
W=> wErrFlw);

fb_ErrPwrMtr(		//Counter errors
	B00:= Power_meter.xErrPwrMtr_1, B01:= Power_meter.xErrPwrMtr_2, B02:= Power_meter.xErrPwrMtr_3,	B03:= Power_meter.xErrPwrMtr_4, 
	B04:= Power_meter.xErrPwrMtr_5, B05:= Power_meter.xErrPwrMtr_6, B06:= Power_meter.xErrPwrMtr_7, B07:= Power_meter.xErrPwrMtr_8, 
	B08:= Power_meter.xErrPwrMtr_9, B09:= Power_meter.xErrPwrMtr_10, B10:= Power_meter.xErrPwrMtr_11, B11:= Power_meter.xErrPwrMtr_12, 
	B12:= Power_meter.xErrPwrMtr_13, B13:= Power_meter.xErrPwrMtr_14, 
W=> wErrPwrMtr);

fb_errothr(			//Misc. errors
	B00:= NOT xVolEn, B01:= xDoor1, B02:= xBattLow, 
W=> wErrOthr);

//xErrorAccum:= (wErrTmp_1 OR wErrTmp_2 OR wErrPrs OR wErrLvl OR wErrFlw OR wErrPwrMtr)>0; //Обобщенные ошибки
          
END_PROGRAM

PROGRAM Main
  VAR
    q_RUN_PLC : PLC_R_STATUS;
  END_VAR

(* CFC diagram, written out as Structured Text *)
(* Выставляем бит работы ПЛК *)
q_RUN_PLC := PLC_R;
xPLC_RUN := 16#002 = q_RUN_PLC;
END_PROGRAM

PROGRAM AI
  VAR
    iTmpRaw_1 AT %MW41420 : INT;
    iTmpRaw_2 AT %MW41421 : INT;
    iTmpRaw_3 AT %MW41422 : INT;
    iTmpRaw_4 AT %MW41423 : INT;
    iTmpRaw_5 AT %MW41424 : INT;
    iTmpRaw_6 AT %MW41425 : INT;
    iTmpRaw_7 AT %MW41426 : INT;
    iTmpRaw_8 AT %MW41427 : INT;
    iTmpRaw_9 AT %MW41428 : INT;
    iTmpRaw_10 AT %MW41429 : INT;
    iTmpRaw_11 AT %MW41430 : INT;
    iTmpRaw_12 AT %MW41431 : INT;
    iTmpRaw_13 AT %MW41432 : INT;
    iTmpRaw_14 AT %MW41433 : INT;
    iTmpRaw_15 AT %MW41434 : INT;
    iTmpRaw_16 AT %MW41435 : INT;
    iTmpRaw_17 AT %MW41436 : INT;
    iTmpRaw_18 AT %MW41437 : INT;
    iTmpRaw_19 AT %MW41438 : INT;
    iTmpRaw_20 AT %MW41439 : INT;
    iTmpRaw_21 AT %MW41440 : INT;
    iTmpRaw_22 AT %MW41441 : INT;
    iTmpRaw_23 AT %MW41442 : INT;
    iTmpRaw_24 AT %MW41443 : INT;
    iTmpRaw_25 AT %MW41444 : INT;
    iTmpRaw_26 AT %MW41445 : INT;
    iTmpRaw_27 AT %MW41446 : INT;
    iTmpRaw_28 AT %MW41447 : INT;
    iTmpRaw_29 AT %MW41448 : INT;
    iTmpRaw_30 AT %MW41449 : INT;
    rTmp_1 AT %MD20010 : REAL;  (* Температура 1 *)
    rTmp_2 AT %MD20011 : REAL;  (* Температура 2 *)
    rTmp_3 AT %MD20012 : REAL;  (* Температура 3 *)
    rTmp_4 AT %MD20013 : REAL;  (* Температура 4 *)
    rTmp_5 AT %MD20014 : REAL;  (* Температура 5 *)
    rTmp_6 AT %MD20015 : REAL;  (* Температура 6 *)
    rTmp_7 AT %MD20016 : REAL;  (* Температура 7 *)
    rTmp_8 AT %MD20017 : REAL;  (* Температура 8 *)
    rTmp_9 AT %MD20018 : REAL;  (* Температура 9 *)
    rTmp_10 AT %MD20019 : REAL;  (* Температура 10 *)
    rTmp_11 AT %MD20020 : REAL;  (* Температура 11 *)
    rTmp_12 AT %MD20021 : REAL;  (* Температура 12 *)
    rTmp_13 AT %MD20022 : REAL;  (* Температура 13 *)
    rTmp_14 AT %MD20023 : REAL;  (* Температура 14 *)
    rTmp_15 AT %MD20024 : REAL;  (* Температура 15 *)
    rTmp_16 AT %MD20025 : REAL;  (* Температура 16 *)
    rTmp_17 AT %MD20026 : REAL;  (* Температура 17 *)
    rTmp_18 AT %MD20027 : REAL;  (* Температура 18 *)
    rTmp_19 AT %MD20028 : REAL;  (* Температура 19 *)
    rTmp_20 AT %MD20029 : REAL;  (* Температура 20 *)
    rTmp_21 AT %MD20030 : REAL;  (* Температура 21 *)
    rTmp_22 AT %MD20031 : REAL;  (* Температура 22 *)
    rTmp_23 AT %MD20032 : REAL;  (* Температура 23 *)
    rTmp_24 AT %MD20033 : REAL;  (* Температура 24 *)
    rTmp_25 AT %MD20034 : REAL;  (* Температура 25 *)
    rTmp_26 AT %MD20035 : REAL;  (* Температура 26 *)
    rTmp_27 AT %MD20036 : REAL;  (* Температура 27 *)
    rTmp_28 AT %MD20037 : REAL;  (* Температура 28 *)
    rTmp_29 AT %MD20038 : REAL;  (* Температура 29 *)
    rTmp_30 AT %MD20039 : REAL;  (* Температура 30 *)
    rTmpK_1 AT %MD10020 : REAL;  (* Коэффициент К Температура _1 *)
    rTmpB_1 AT %MD10021 : REAL;  (* Коэффициент В Температура _1 *)
    rTmpK_2 AT %MD10022 : REAL;  (* Коэффициент К Температура _2 *)
    rTmpB_2 AT %MD10023 : REAL;  (* Коэффициент В Температура _2 *)
    rTmpK_3 AT %MD10024 : REAL;  (* Коэффициент К Температура _3 *)
    rTmpB_3 AT %MD10025 : REAL;  (* Коэффициент В Температура _3 *)
    rTmpK_4 AT %MD10026 : REAL;  (* Коэффициент К Температура _4 *)
    rTmpB_4 AT %MD10027 : REAL;  (* Коэффициент В Температура _4 *)
    rTmpK_5 AT %MD10028 : REAL;  (* Коэффициент К Температура _5 *)
    rTmpB_5 AT %MD10029 : REAL;  (* Коэффициент В Температура _5 *)
    rTmpK_6 AT %MD10030 : REAL;  (* Коэффициент К Температура _6 *)
    rTmpB_6 AT %MD10031 : REAL;  (* Коэффициент В Температура _6 *)
    rTmpK_7 AT %MD10032 : REAL;  (* Коэффициент К Температура _7 *)
    rTmpB_7 AT %MD10033 : REAL;  (* Коэффициент В Температура _7 *)
    rTmpK_8 AT %MD10034 : REAL;  (* Коэффициент К Температура _8 *)
    rTmpB_8 AT %MD10035 : REAL;  (* Коэффициент В Температура _8 *)
    rTmpK_9 AT %MD10036 : REAL;  (* Коэффициент К Температура _9 *)
    rTmpB_9 AT %MD10037 : REAL;  (* Коэффициент В Температура _9 *)
    rTmpK_10 AT %MD10038 : REAL;  (* Коэффициент К Температура _10 *)
    rTmpB_10 AT %MD10039 : REAL;  (* Коэффициент В Температура _10 *)
    rTmpK_11 AT %MD10040 : REAL;  (* Коэффициент К Температура _11 *)
    rTmpB_11 AT %MD10041 : REAL;  (* Коэффициент В Температура _11 *)
    rTmpK_12 AT %MD10042 : REAL;  (* Коэффициент К Температура _12 *)
    rTmpB_12 AT %MD10043 : REAL;  (* Коэффициент В Температура _12 *)
    rTmpK_13 AT %MD10044 : REAL;  (* Коэффициент К Температура _13 *)
    rTmpB_13 AT %MD10045 : REAL;  (* Коэффициент В Температура _13 *)
    rTmpK_14 AT %MD10046 : REAL;  (* Коэффициент К Температура _14 *)
    rTmpB_14 AT %MD10047 : REAL;  (* Коэффициент В Температура _14 *)
    rTmpK_15 AT %MD10048 : REAL;  (* Коэффициент К Температура _15 *)
    rTmpB_15 AT %MD10049 : REAL;  (* Коэффициент В Температура _15 *)
    rTmpK_16 AT %MD10050 : REAL;  (* Коэффициент К Температура _16 *)
    rTmpB_16 AT %MD10051 : REAL;  (* Коэффициент В Температура _16 *)
    rTmpK_17 AT %MD10052 : REAL;  (* Коэффициент К Температура _17 *)
    rTmpB_17 AT %MD10053 : REAL;  (* Коэффициент В Температура _17 *)
    rTmpK_18 AT %MD10054 : REAL;  (* Коэффициент К Температура _18 *)
    rTmpB_18 AT %MD10055 : REAL;  (* Коэффициент В Температура _18 *)
    rTmpK_19 AT %MD10056 : REAL;  (* Коэффициент К Температура _19 *)
    rTmpB_19 AT %MD10057 : REAL;  (* Коэффициент В Температура _19 *)
    rTmpK_20 AT %MD10058 : REAL;  (* Коэффициент К Температура _20 *)
    rTmpB_20 AT %MD10059 : REAL;  (* Коэффициент В Температура _20 *)
    rTmpK_21 AT %MD10060 : REAL;  (* Коэффициент К Температура _21 *)
    rTmpB_21 AT %MD10061 : REAL;  (* Коэффициент В Температура _21 *)
    rTmpK_22 AT %MD10062 : REAL;  (* Коэффициент К Температура _22 *)
    rTmpB_22 AT %MD10063 : REAL;  (* Коэффициент В Температура _22 *)
    rTmpK_23 AT %MD10064 : REAL;  (* Коэффициент К Температура _23 *)
    rTmpB_23 AT %MD10065 : REAL;  (* Коэффициент В Температура _23 *)
    rTmpK_24 AT %MD10066 : REAL;  (* Коэффициент К Температура _24 *)
    rTmpB_24 AT %MD10067 : REAL;  (* Коэффициент В Температура _24 *)
    rTmpK_25 AT %MD10068 : REAL;  (* Коэффициент К Температура _25 *)
    rTmpB_25 AT %MD10069 : REAL;  (* Коэффициент В Температура _25 *)
    rTmpK_26 AT %MD10070 : REAL;  (* Коэффициент К Температура _26 *)
    rTmpB_26 AT %MD10071 : REAL;  (* Коэффициент В Температура _26 *)
    rTmpK_27 AT %MD10072 : REAL;  (* Коэффициент К Температура _27 *)
    rTmpB_27 AT %MD10073 : REAL;  (* Коэффициент В Температура _27 *)
    rTmpK_28 AT %MD10074 : REAL;  (* Коэффициент К Температура _28 *)
    rTmpB_28 AT %MD10075 : REAL;  (* Коэффициент В Температура _28 *)
    rTmpK_29 AT %MD10076 : REAL;  (* Коэффициент К Температура _29 *)
    rTmpB_29 AT %MD10077 : REAL;  (* Коэффициент В Температура _29 *)
    rTmpK_30 AT %MD10078 : REAL;  (* Коэффициент К Температура _30 *)
    rTmpB_30 AT %MD10079 : REAL;  (* Коэффициент В Температура _30 *)
    iPrsRaw_1 AT %MW41410 : INT;
    iPrsRaw_2 AT %MW41411 : INT;
    iPrsRaw_3 AT %MW41412 : INT;
    iPrsRaw_4 AT %MW41413 : INT;
    iPrsRaw_5 AT %MW41414 : INT;
    iPrsRaw_6 AT %MW41415 : INT;
    iPrsRaw_7 AT %MW41416 : INT;
    iPrsRaw_8 AT %MW41417 : INT;
    iPrsRaw_9 AT %MW41418 : INT;
    iPrsRaw_10 AT %MW41419 : INT;
    rPrs_1 AT %MD20000 : REAL;  (* Давление 1 *)
    rPrs_2 AT %MD20001 : REAL;  (* Давление 2 *)
    rPrs_3 AT %MD20002 : REAL;  (* Давление 3 *)
    rPrs_4 AT %MD20003 : REAL;  (* Давление 4 *)
    rPrs_5 AT %MD20004 : REAL;  (* Давление 5 *)
    rPrs_6 AT %MD20005 : REAL;  (* Давление 6 *)
    rPrs_7 AT %MD20006 : REAL;  (* Давление 7 *)
    rPrs_8 AT %MD20007 : REAL;  (* Давление 8 *)
    rPrs_9 AT %MD20008 : REAL;  (* Давление 9 *)
    rPrs_10 AT %MD20009 : REAL;  (* Давление 10 *)
    rPrsK_1 AT %MD10000 : REAL;  (* Коэффициент К Давление 1 *)
    rPrsB_1 AT %MD10001 : REAL;  (* Коэффициент В Давление 1 *)
    rPrsK_2 AT %MD10002 : REAL;  (* Коэффициент К Давление 2 *)
    rPrsB_2 AT %MD10003 : REAL;  (* Коэффициент В Давление 2 *)
    rPrsK_3 AT %MD10004 : REAL;  (* Коэффициент К Давление 3 *)
    rPrsB_3 AT %MD10005 : REAL;  (* Коэффициент В Давление 3 *)
    rPrsK_4 AT %MD10006 : REAL;  (* Коэффициент К Давление 4 *)
    rPrsB_4 AT %MD10007 : REAL;  (* Коэффициент В Давление 4 *)
    rPrsK_5 AT %MD10008 : REAL;  (* Коэффициент К Давление 5 *)
    rPrsB_5 AT %MD10009 : REAL;  (* Коэффициент В Давление 5 *)
    rPrsK_6 AT %MD10010 : REAL;  (* Коэффициент К Давление 6 *)
    rPrsB_6 AT %MD10011 : REAL;  (* Коэффициент В Давление 6 *)
    rPrsK_7 AT %MD10012 : REAL;  (* Коэффициент К Давление 7 *)
    rPrsB_7 AT %MD10013 : REAL;  (* Коэффициент В Давление 7 *)
    rPrsK_8 AT %MD10014 : REAL;  (* Коэффициент К Давление 8 *)
    rPrsB_8 AT %MD10015 : REAL;  (* Коэффициент В Давление 8 *)
    rPrsK_9 AT %MD10016 : REAL;  (* Коэффициент К Давление 9 *)
    rPrsB_9 AT %MD10017 : REAL;  (* Коэффициент В Давление 9 *)
    rPrsK_10 AT %MD10018 : REAL;  (* Коэффициент К Давление 10 *)
    rPrsB_10 AT %MD10019 : REAL;  (* Коэффициент В Давление 10 *)
    iLvlRaw_1 AT %MW41450 : INT;
    iLvlRaw_2 AT %MW41451 : INT;
    iLvlRaw_3 AT %MW41452 : INT;
    iLvlRaw_4 AT %MW41453 : INT;
    iLvlRaw_5 AT %MW41454 : INT;
    iLvlRaw_6 AT %MW41455 : INT;
    rLvl_1 AT %MD20040 : REAL;  (* Уровень 1 *)
    rLvl_2 AT %MD20041 : REAL;  (* Уровень 2 *)
    rLvl_3 AT %MD20042 : REAL;  (* Уровень 3 *)
    rLvl_4 AT %MD20043 : REAL;  (* Уровень 4 *)
    rLvl_5 AT %MD20044 : REAL;  (* Уровень 5 *)
    rLvl_6 AT %MD20045 : REAL;  (* Уровень 6 *)
    rLvlK_1 AT %MD10080 : REAL;  (* Коэффициент К Уровень 1 *)
    rLvlB_1 AT %MD10081 : REAL;  (* Коэффициент В Уровень 1 *)
    rLvlK_2 AT %MD10082 : REAL;  (* Коэффициент К Уровень 2 *)
    rLvlB_2 AT %MD10083 : REAL;  (* Коэффициент В Уровень 2 *)
    rLvlK_3 AT %MD10084 : REAL;  (* Коэффициент К Уровень 3 *)
    rLvlB_3 AT %MD10085 : REAL;  (* Коэффициент В Уровень 3 *)
    rLvlK_4 AT %MD10086 : REAL;  (* Коэффициент К Уровень 4 *)
    rLvlB_4 AT %MD10087 : REAL;  (* Коэффициент В Уровень 4 *)
    rLvlK_5 AT %MD10088 : REAL;  (* Коэффициент К Уровень 5 *)
    rLvlB_5 AT %MD10089 : REAL;  (* Коэффициент В Уровень 5 *)
    rLvlK_6 AT %MD10090 : REAL;  (* Коэффициент К Уровень 6 *)
    rLvlB_6 AT %MD10091 : REAL;  (* Коэффициент В Уровень 6 *)
  END_VAR
  VAR
    fb_Tmp_1 : Analog_Input;
    fb_Tmp_2 : Analog_Input;
    fb_Tmp_3 : Analog_Input;
    fb_Tmp_4 : Analog_Input;
    fb_Tmp_5 : Analog_Input;
    fb_Tmp_6 : Analog_Input;
    fb_Tmp_7 : Analog_Input;
    fb_Tmp_8 : Analog_Input;
    fb_Tmp_9 : Analog_Input;
    fb_Tmp_10 : Analog_Input;
    fb_Tmp_11 : Analog_Input;
    fb_Tmp_12 : Analog_Input;
    fb_Tmp_13 : Analog_Input;
    fb_Tmp_14 : Analog_Input;
    fb_Tmp_15 : Analog_Input;
    fb_Tmp_16 : Analog_Input;
    fb_Tmp_17 : Analog_Input;
    fb_Tmp_18 : Analog_Input;
    fb_Tmp_19 : Analog_Input;
    fb_Tmp_20 : Analog_Input;
    fb_Tmp_21 : Analog_Input;
    fb_Tmp_22 : Analog_Input;
    fb_Tmp_23 : Analog_Input;
    fb_Tmp_24 : Analog_Input;
    fb_Tmp_25 : Analog_Input;
    fb_Tmp_26 : Analog_Input;
    fb_Tmp_27 : Analog_Input;
    fb_Tmp_28 : Analog_Input;
    fb_Tmp_29 : Analog_Input;
    fb_Tmp_30 : Analog_Input;
    fb_Prs_1 : Analog_Input;
    fb_Prs_2 : Analog_Input;
    fb_Prs_3 : Analog_Input;
    fb_Prs_4 : Analog_Input;
    fb_Prs_5 : Analog_Input;
    fb_Prs_6 : Analog_Input;
    fb_Lvl_1 : Analog_Input;
    fb_Lvl_2 : Analog_Input;
    fb_Lvl_3 : Analog_Input;
    fb_Lvl_4 : Analog_Input;
    fb_Lvl_5 : Analog_Input;
    fb_Lvl_6 : Analog_Input;
    bErrTmp_1 : BYTE;
    bErrTmp_2 : BYTE;
    bErrTmp_3 : BYTE;
    bErrTmp_4 : BYTE;
    bErrTmp_5 : BYTE;
    bErrTmp_6 : BYTE;
    bErrTmp_7 : BYTE;
    bErrTmp_8 : BYTE;
    bErrTmp_9 : BYTE;
    bErrTmp_10 : BYTE;
    bErrTmp_11 : BYTE;
    bErrTmp_12 : BYTE;
    bErrTmp_13 : BYTE;
    bErrTmp_14 : BYTE;
    bErrTmp_15 : BYTE;
    bErrTmp_16 : BYTE;
    bErrTmp_17 : BYTE;
    bErrTmp_18 : BYTE;
    bErrTmp_19 : BYTE;
    bErrTmp_20 : BYTE;
    bErrTmp_21 : BYTE;
    bErrTmp_22 : BYTE;
    bErrTmp_23 : BYTE;
    bErrTmp_24 : BYTE;
    bErrTmp_25 : BYTE;
    bErrTmp_26 : BYTE;
    bErrTmp_27 : BYTE;
    bErrTmp_28 : BYTE;
    bErrTmp_29 : BYTE;
    bErrTmp_30 : BYTE;
    bErrPrs_1 : BYTE;
    bErrPrs_2 : BYTE;
    bErrPrs_3 : BYTE;
    bErrPrs_4 : BYTE;
    bErrPrs_5 : BYTE;
    bErrPrs_6 : BYTE;
    bErrLvl_1 : BYTE;
    bErrLvl_2 : BYTE;
    bErrLvl_3 : BYTE;
    bErrLvl_4 : BYTE;
    bErrLvl_5 : BYTE;
    bErrLvl_6 : BYTE;
    xErrPrs_1 : BOOL;
    xErrPrs_2 : BOOL;
    xErrPrs_3 : BOOL;
    xErrPrs_4 : BOOL;
    xErrPrs_5 : BOOL;
    xErrPrs_6 : BOOL;
    xErrTmp_1 : BOOL;
    xErrTmp_2 : BOOL;
    xErrTmp_3 : BOOL;
    xErrTmp_4 : BOOL;
    xErrTmp_5 : BOOL;
    xErrTmp_6 : BOOL;
    xErrTmp_7 : BOOL;
    xErrTmp_8 : BOOL;
    xErrTmp_9 : BOOL;
    xErrTmp_10 : BOOL;
    xErrTmp_11 : BOOL;
    xErrTmp_12 : BOOL;
    xErrTmp_13 : BOOL;
    xErrTmp_14 : BOOL;
    xErrTmp_15 : BOOL;
    xErrTmp_16 : BOOL;
    xErrTmp_17 : BOOL;
    xErrTmp_18 : BOOL;
    xErrTmp_19 : BOOL;
    xErrTmp_20 : BOOL;
    xErrTmp_21 : BOOL;
    xErrTmp_22 : BOOL;
    xErrTmp_23 : BOOL;
    xErrTmp_24 : BOOL;
    xErrTmp_25 : BOOL;
    xErrTmp_26 : BOOL;
    xErrTmp_27 : BOOL;
    xErrTmp_28 : BOOL;
    xErrTmp_29 : BOOL;
    xErrTmp_30 : BOOL;
    xErrLvl_1 : BOOL;
    xErrLvl_2 : BOOL;
    xErrLvl_3 : BOOL;
    xErrLvl_4 : BOOL;
    xErrLvl_5 : BOOL;
    xErrLvl_6 : BOOL;
  END_VAR

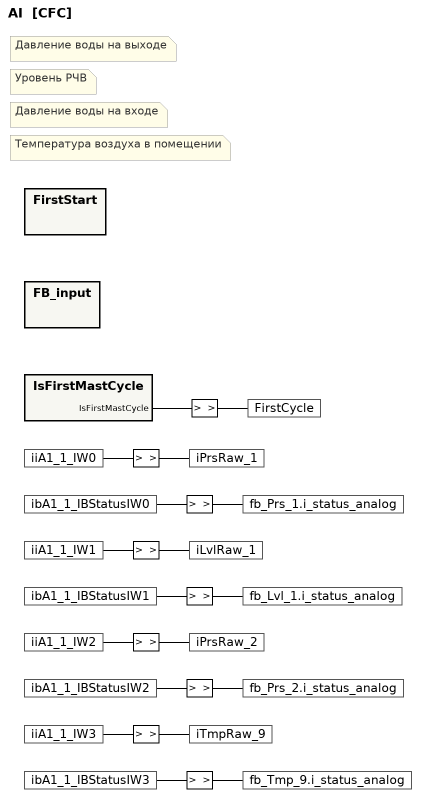
(* CFC diagram, written out as Structured Text *)
(* Давление воды на выходе *)
FirstStart();
FB_input();
(* Уровень РЧВ *)
iPrsRaw_1 := iiA1_1_IW0;
(* Давление воды на входе *)
fb_Prs_1.i_status_analog := ibA1_1_IBStatusIW0;
FirstCycle := IsFirstMastCycle();
iLvlRaw_1 := iiA1_1_IW1;
(* Температура воздуха в помещении *)
fb_Lvl_1.i_status_analog := ibA1_1_IBStatusIW1;
iPrsRaw_2 := iiA1_1_IW2;
fb_Prs_2.i_status_analog := ibA1_1_IBStatusIW2;
iTmpRaw_9 := iiA1_1_IW3;
fb_Tmp_9.i_status_analog := ibA1_1_IBStatusIW3;

ACTION FirstStart:
                IF FirstCycle THEN
(*rTmpK_1:=0;
rTmpB_1:=0;
rTmpK_2:=0;
rTmpB_2:=0;
rTmpK_3:=0;
rTmpB_3:=0;
rTmpK_4:=0;
rTmpB_4:=0;
rTmpK_5:=0;
rTmpB_5:=0;
rTmpK_6:=0;
rTmpB_6:=0;
rTmpK_7:=0;
rTmpB_7:=0;
rTmpK_8:=0;
rTmpB_8:=0;*)
rTmpK_9:=1000;		//Температура воздуха в помещении
rTmpB_9:=0;
rTmpK_10:=100; 		//Температура воздуха в помещении
rTmpB_10:=0;(*
rTmpK_11:=0;
rTmpB_11:=0;
rTmpK_12:=0;
rTmpB_12:=0;
rTmpK_13:=0;
rTmpB_13:=0;
rTmpK_14:=0;
rTmpB_14:=0;
rTmpK_15:=0;
rTmpB_15:=0;
rTmpK_16:=0;
rTmpB_16:=0;
*)
rPrsK_1:=16;		//Давление воды 
rPrsB_1:=0;
rPrsK_2:=16;
rPrsB_2:=0;
rPrsK_3:=16;
rPrsB_3:=0;
rPrsK_4:=16;
rPrsB_4:=0;
rPrsK_5:=16;
rPrsB_5:=0;
rPrsK_6:=16;
rPrsB_6:=0;

rLvlK_1:=5;
rLvlB_1:=0;
rLvlK_2:=5;
rLvlB_2:=0;(*
rLvlK_3:=0;
rLvlB_3:=0;*)
END_IF;
              
END_ACTION

ACTION FB_input:
                fb_Tmp_1(
	i_sensor_value:= iTmpRaw_1, 
	k:= rTmpK_1, b:= rTmpB_1, i_ADC_Range:= i_ADC_Range, 
	q_status_analog=> bErrTmp_1, xAlarm_bit=> xErrTmp_1,
	q_Out=> rTmp_1, );
fb_Tmp_2(
	i_sensor_value:= iTmpRaw_2, 
	k:= rTmpK_2, b:= rTmpB_2, i_ADC_Range:= i_ADC_Range, 
	q_status_analog=> bErrTmp_2, xAlarm_bit=> xErrTmp_2,
	q_Out=> rTmp_2, );
fb_Tmp_3(
	i_sensor_value:= iTmpRaw_3, 
	k:= rTmpK_3, b:= rTmpB_3, i_ADC_Range:= i_ADC_Range, 
	q_status_analog=> bErrTmp_3, xAlarm_bit=> xErrTmp_3,
	q_Out=> rTmp_3, );
fb_Tmp_4(
	i_sensor_value:= iTmpRaw_4, 
	k:= rTmpK_4, b:= rTmpB_4, i_ADC_Range:= i_ADC_Range, 
	q_status_analog=> bErrTmp_4, xAlarm_bit=> xErrTmp_4,
	q_Out=> rTmp_4, );
fb_Tmp_5(
	i_sensor_value:= iTmpRaw_5, 
	k:= rTmpK_5, b:= rTmpB_5, i_ADC_Range:= i_ADC_Range, 
	q_status_analog=> bErrTmp_5, xAlarm_bit=> xErrTmp_5,
	q_Out=> rTmp_5, );
fb_Tmp_6(
	i_sensor_value:= iTmpRaw_6, 
	k:= rTmpK_6, b:= rTmpB_6, i_ADC_Range:= i_ADC_Range, 
	q_status_analog=> bErrTmp_6, xAlarm_bit=> xErrTmp_6,
	q_Out=> rTmp_6, );
fb_Tmp_7(
	i_sensor_value:= iTmpRaw_7, 
	k:= rTmpK_7, b:= rTmpB_7, i_ADC_Range:= i_ADC_Range, 
	q_status_analog=> bErrTmp_7, xAlarm_bit=> xErrTmp_7,
	q_Out=> rTmp_7, );
fb_Tmp_8(
	i_sensor_value:= iTmpRaw_8, 
	k:= rTmpK_8, b:= rTmpB_8, i_ADC_Range:= i_ADC_Range, 
	q_status_analog=> bErrTmp_8, xAlarm_bit=> xErrTmp_8,
	q_Out=> rTmp_8, );
fb_Tmp_9(
	i_sensor_value:= iTmpRaw_9, 
	k:= rTmpK_9, b:= rTmpB_9, i_ADC_Range:= i_ADC_Range, 
	q_status_analog=> bErrTmp_9, xAlarm_bit=> xErrTmp_9,
	q_Out=> rTmp_9, );
fb_Tmp_10(
	i_sensor_value:= iTmpRaw_10, 
	k:= rTmpK_10, b:= rTmpB_10, i_ADC_Range:= i_ADC_Range, 
	q_status_analog=> bErrTmp_10, xAlarm_bit=> xErrTmp_10,
	q_Out=> rTmp_10, );
fb_Tmp_11(
	i_sensor_value:= iTmpRaw_11, 
	k:= rTmpK_11, b:= rTmpB_11, i_ADC_Range:= i_ADC_Range, 
	q_status_analog=> bErrTmp_11, xAlarm_bit=> xErrTmp_11,
	q_Out=> rTmp_11, );
fb_Tmp_12(
	i_sensor_value:= iTmpRaw_12, 
	k:= rTmpK_12, b:= rTmpB_12, i_ADC_Range:= i_ADC_Range, 
	q_status_analog=> bErrTmp_12, xAlarm_bit=> xErrTmp_12,
	q_Out=> rTmp_12, );
fb_Tmp_13(
	i_sensor_value:= iTmpRaw_13, 
	k:= rTmpK_13, b:= rTmpB_13, i_ADC_Range:= i_ADC_Range, 
	q_status_analog=> bErrTmp_13, xAlarm_bit=> xErrTmp_13,
	q_Out=> rTmp_13, );
fb_Tmp_14(
	i_sensor_value:= iTmpRaw_14, 
	k:= rTmpK_14, b:= rTmpB_14, i_ADC_Range:= i_ADC_Range, 
	q_status_analog=> bErrTmp_14, xAlarm_bit=> xErrTmp_14,
	q_Out=> rTmp_14, );
fb_Tmp_15(
	i_sensor_value:= iTmpRaw_15, 
	k:= rTmpK_15, b:= rTmpB_15, i_ADC_Range:= i_ADC_Range, 
	q_status_analog=> bErrTmp_15, xAlarm_bit=> xErrTmp_15,
	q_Out=> rTmp_15, );
fb_Tmp_16(
	i_sensor_value:= iTmpRaw_16, 
	k:= rTmpK_16, b:= rTmpB_16, i_ADC_Range:= i_ADC_Range, 
	q_status_analog=> bErrTmp_16, xAlarm_bit=> xErrTmp_16,
	q_Out=> rTmp_16, );
fb_Tmp_17(
	i_sensor_value:= iTmpRaw_17, 
	k:= rTmpK_17, b:= rTmpB_17, i_ADC_Range:= i_ADC_Range, 
	q_status_analog=> bErrTmp_17, xAlarm_bit=> xErrTmp_17,
	q_Out=> rTmp_17, );
fb_Tmp_18(
	i_sensor_value:= iTmpRaw_18, 
	k:= rTmpK_18, b:= rTmpB_18, i_ADC_Range:= i_ADC_Range, 
	q_status_analog=> bErrTmp_18, xAlarm_bit=> xErrTmp_18,
	q_Out=> rTmp_18, );
fb_Tmp_19(
	i_sensor_value:= iTmpRaw_19, 
	k:= rTmpK_19, b:= rTmpB_19, i_ADC_Range:= i_ADC_Range, 
	q_status_analog=> bErrTmp_19, xAlarm_bit=> xErrTmp_19,
	q_Out=> rTmp_19, );
fb_Tmp_20(
	i_sensor_value:= iTmpRaw_20, 
	k:= rTmpK_20, b:= rTmpB_20, i_ADC_Range:= i_ADC_Range, 
	q_status_analog=> bErrTmp_20, xAlarm_bit=> xErrTmp_20,
	q_Out=> rTmp_20, );
fb_Tmp_21(
	i_sensor_value:= iTmpRaw_21, 
	k:= rTmpK_21, b:= rTmpB_21, i_ADC_Range:= i_ADC_Range, 
	q_status_analog=> bErrTmp_21, xAlarm_bit=> xErrTmp_21,
	q_Out=> rTmp_21, );
fb_Tmp_22(
	i_sensor_value:= iTmpRaw_22, 
	k:= rTmpK_22, b:= rTmpB_22, i_ADC_Range:= i_ADC_Range, 
	q_status_analog=> bErrTmp_22, xAlarm_bit=> xErrTmp_22,
	q_Out=> rTmp_22, );
fb_Tmp_23(
	i_sensor_value:= iTmpRaw_23, 
	k:= rTmpK_23, b:= rTmpB_23, i_ADC_Range:= i_ADC_Range, 
	q_status_analog=> bErrTmp_23, xAlarm_bit=> xErrTmp_23,
	q_Out=> rTmp_23, );
fb_Tmp_24(
	i_sensor_value:= iTmpRaw_24, 
	k:= rTmpK_24, b:= rTmpB_24, i_ADC_Range:= i_ADC_Range, 
	q_status_analog=> bErrTmp_24, xAlarm_bit=> xErrTmp_24,
	q_Out=> rTmp_24, );
fb_Tmp_25(
	i_sensor_value:= iTmpRaw_25, 
	k:= rTmpK_25, b:= rTmpB_25, i_ADC_Range:= i_ADC_Range, 
	q_status_analog=> bErrTmp_25, xAlarm_bit=> xErrTmp_25,
	q_Out=> rTmp_25, );
fb_Tmp_26(
	i_sensor_value:= iTmpRaw_26, 
	k:= rTmpK_26, b:= rTmpB_26, i_ADC_Range:= i_ADC_Range, 
	q_status_analog=> bErrTmp_26, xAlarm_bit=> xErrTmp_26,
	q_Out=> rTmp_26, );
fb_Tmp_27(
	i_sensor_value:= iTmpRaw_27, 
	k:= rTmpK_27, b:= rTmpB_27, i_ADC_Range:= i_ADC_Range, 
	q_status_analog=> bErrTmp_27, xAlarm_bit=> xErrTmp_27,
	q_Out=> rTmp_27, );
fb_Tmp_28(
	i_sensor_value:= iTmpRaw_28, 
	k:= rTmpK_28, b:= rTmpB_28, i_ADC_Range:= i_ADC_Range, 
	q_status_analog=> bErrTmp_28, xAlarm_bit=> xErrTmp_28,
	q_Out=> rTmp_28, );
fb_Tmp_29(
	i_sensor_value:= iTmpRaw_29, 
	k:= rTmpK_29, b:= rTmpB_29, i_ADC_Range:= i_ADC_Range, 
	q_status_analog=> bErrTmp_29, xAlarm_bit=> xErrTmp_29,
	q_Out=> rTmp_29, );
fb_Tmp_30(
	i_sensor_value:= iTmpRaw_30, 
	k:= rTmpK_30, b:= rTmpB_30, i_ADC_Range:= i_ADC_Range, 
	q_status_analog=> bErrTmp_30, xAlarm_bit=> xErrTmp_30,
	q_Out=> rTmp_30, );
fb_Prs_1(
	i_sensor_value:= iPrsRaw_1, 
	k:= rPrsK_1*1.0197, b:= rPrsB_1, i_ADC_Range:= i_ADC_Range, 
	q_status_analog=> bErrPrs_1, xAlarm_bit=> xErrPrs_1,
	q_Out=> rPrs_1, );
fb_Prs_2(
	i_sensor_value:= iPrsRaw_2, 
	k:= rPrsK_2*1.0197, b:= rPrsB_2, i_ADC_Range:= i_ADC_Range, 
	q_status_analog=> bErrPrs_2, xAlarm_bit=> xErrPrs_2,
	q_Out=> rPrs_2, );
fb_Prs_3(
	i_sensor_value:= iPrsRaw_3, 
	k:= rPrsK_3*1.0197, b:= rPrsB_3, i_ADC_Range:= i_ADC_Range, 
	q_status_analog=> bErrPrs_3, xAlarm_bit=> xErrPrs_3,
	q_Out=> rPrs_3, );
fb_Prs_4(
	i_sensor_value:= iPrsRaw_4, 
	k:= rPrsK_4*1.0197, b:= rPrsB_4, i_ADC_Range:= i_ADC_Range, 
	q_status_analog=> bErrPrs_4, xAlarm_bit=> xErrPrs_4,
	q_Out=> rPrs_4, );
fb_Prs_5(
	i_sensor_value:= iPrsRaw_5, 
	k:= rPrsK_5, b:= rPrsB_5, i_ADC_Range:= i_ADC_Range, 
	q_status_analog=> bErrPrs_5, xAlarm_bit=> xErrPrs_5,
	q_Out=> rPrs_5, );
fb_Prs_6(
	i_sensor_value:= iPrsRaw_6, 
	k:= rPrsK_6, b:= rPrsB_6, i_ADC_Range:= i_ADC_Range, 
	q_status_analog=> bErrPrs_6, xAlarm_bit=> xErrPrs_6,
	q_Out=> rPrs_6, );
fb_Lvl_1(
	i_sensor_value:= iLvlRaw_1, 
	k:= rLvlK_1, b:= rLvlB_1, i_ADC_Range:= i_ADC_Range, 
	q_status_analog=> bErrLvl_1, xAlarm_bit=> xErrLvl_1,
	q_Out=> rLvl_1, );
fb_Lvl_2(
	i_sensor_value:= iLvlRaw_2, 
	k:= rLvlK_2, b:= rLvlB_2, i_ADC_Range:= i_ADC_Range, 
	q_status_analog=> bErrLvl_2, xAlarm_bit=> xErrLvl_2,
	q_Out=> rLvl_2, );
fb_Lvl_3(
	i_sensor_value:= iLvlRaw_3, 
	k:= rLvlK_3, b:= rLvlB_3, i_ADC_Range:= i_ADC_Range, 
	q_status_analog=> bErrLvl_3, xAlarm_bit=> xErrLvl_3,
	q_Out=> rLvl_3, );
fb_Lvl_4(
	i_sensor_value:= iLvlRaw_4, 
	k:= rLvlK_4, b:= rLvlB_4, i_ADC_Range:= i_ADC_Range, 
	q_status_analog=> bErrLvl_4, xAlarm_bit=> xErrLvl_4,
	q_Out=> rLvl_4, );
fb_Lvl_5(
	i_sensor_value:= iLvlRaw_5, 
	k:= rLvlK_5, b:= rLvlB_5, i_ADC_Range:= i_ADC_Range, 
	q_status_analog=> bErrLvl_5, xAlarm_bit=> xErrLvl_5,
	q_Out=> rLvl_5, );
fb_Lvl_6(
	i_sensor_value:= iLvlRaw_6, 
	k:= rLvlK_6, b:= rLvlB_6, i_ADC_Range:= i_ADC_Range, 
	q_status_analog=> bErrLvl_6, xAlarm_bit=> xErrLvl_6,
	q_Out=> rLvl_6, );

              
END_ACTION
END_PROGRAM

PROGRAM D_input
  VAR
    wDI_int AT %MW41012 : WORD;
  END_VAR

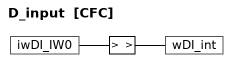
(* CFC diagram, written out as Structured Text *)
wDI_int := iwDI_IW0;
END_PROGRAM

PROGRAM D_output
  VAR
    d_out : BIT_AS_WORD;
  END_VAR

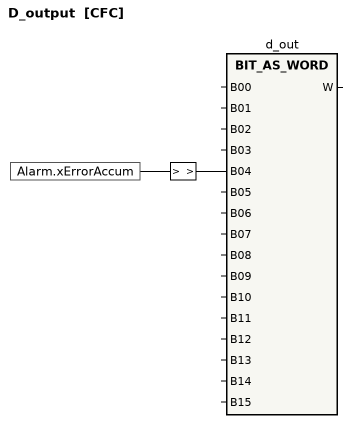
(* CFC diagram, written out as Structured Text *)
d_out(B04 := Alarm.xErrorAccum);
END_PROGRAM

(* Implicitly generated code : DO NOT EDIT *)
{attribute 'check_bounds'}
{attribute 'no_check'}
FUNCTION CheckBounds : DINT
  VAR_INPUT
    index : DINT;
    lower : DINT;
    upper : DINT;
  END_VAR

            // Implicitly generated code : Only an Implementation suggestion
IF  index < lower THEN
	CheckBounds := lower;
ELSIF  index > upper THEN
	CheckBounds := upper;
ELSE  
	CheckBounds := index;
END_IF

          
END_FUNCTION

FUNCTION_BLOCK Comm_error
  VAR_INPUT
    i_comm_error : INT;
  END_VAR
  VAR_OUTPUT
    q_alarm_comm : BOOL;
    q_set_measurment : BOOL;
  END_VAR
  VAR
    CTU_0 : CTU;
    SR_1 : SR;
    TON_1 : TON;
    R_TRIG_0 : R_TRIG;
    TON_2 : TON;
    R_TRIG_1 : R_TRIG;
    TP_1 : TP;
    RS_1 : RS;
    TON_3 : TON;
  END_VAR
  VAR  (* added by the conversion: wires and edge detectors of the diagram *)
    _OR35_OUT : BOOL;
    _GT7_OUT : BOOL;
  END_VAR

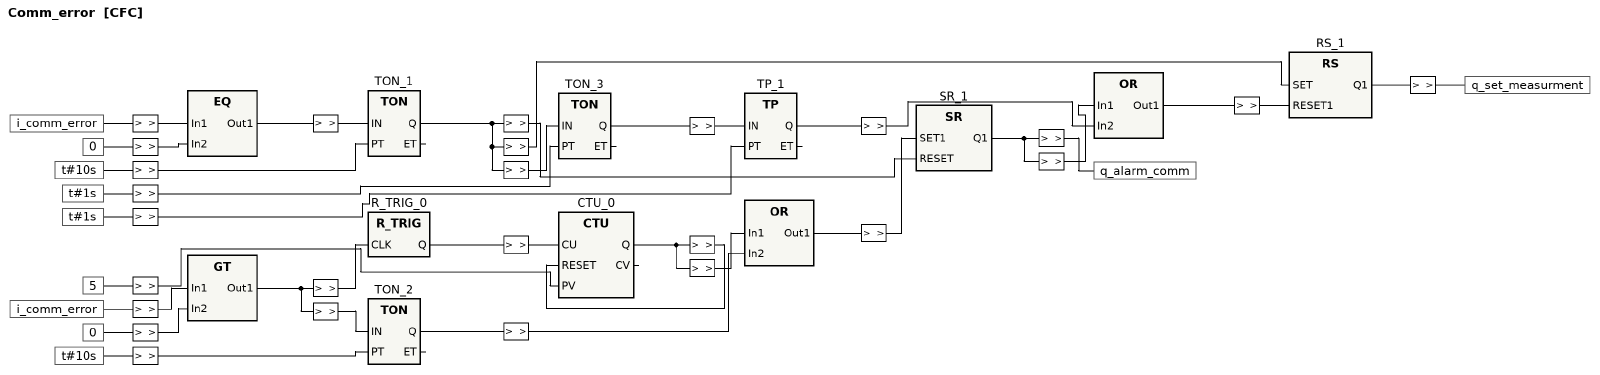
(* CFC diagram, written out as Structured Text *)
RS_1(SET := TON_1.Q, RESET1 := _OR35_OUT);
_GT7_OUT := i_comm_error > 0;
R_TRIG_0(CLK := _GT7_OUT);
CTU_0(CU := R_TRIG_0.Q, RESET := CTU_0.Q, PV := 5);
TON_2(IN := _GT7_OUT, PT := t#10s);
TON_1(IN := i_comm_error = 0, PT := t#10s);
SR_1(SET1 := CTU_0.Q OR TON_2.Q, RESET := TON_1.Q);
q_alarm_comm := SR_1.Q1;
TON_3(IN := TON_1.Q, PT := t#1s);
_OR35_OUT := SR_1.Q1 OR TP_1.Q;
TP_1(IN := TON_3.Q, PT := t#1s);
q_set_measurment := RS_1.Q1;
END_FUNCTION_BLOCK

FUNCTION_BLOCK Stat_to_num
  VAR_INPUT
    in0 : BOOL;
    in1 : BOOL;
    in2 : BOOL;
    in3 : BOOL;
    in4 : BOOL;
    in5 : BOOL;
    in6 : BOOL;
    in7 : BOOL;
  END_VAR
  VAR
    selectors : ARRAY[0..7] OF BOOL;
    i : BYTE;
    chk : BOOL;
  END_VAR
  VAR_OUTPUT
    out : WORD;
  END_VAR

            selectors[0]:=in0;
selectors[1]:=in1;
selectors[2]:=in2;
selectors[3]:=in3;
selectors[4]:=in4;
selectors[5]:=in5;
selectors[6]:=in6;
selectors[7]:=in7;

IF chk THEN
	chk:=0;
ELSE
	out:=0;
END_IF;
FOR i:=0 TO 7 BY 1 DO
	IF selectors[i] THEN
		out:=i;
		chk:=1;
	END_IF;
END_FOR;
          
END_FUNCTION_BLOCK

